(* CODESYS project plc_eposcmd.library
   Company: Maxon Motor
   Title: Maxon
   Version: 1.0.0.0

Project tree, tasks and I/O mapping:
  libraries: Tc2_System, * (Beckhoff Automation GmbH); Tc2_Standard, * (Beckhoff Automation GmbH)
  Data types/
  Global Variables/
    global variables Globale_Variablen
  POUs/
    Configuration/
      function block FB_GetCurrentRegulatorGain [ST]
      function block FB_GetEncoderParameter [ST]
      function block FB_GetMotorParameter [ST]
      function block FB_GetPositionRegulatorGain [ST]
      function block FB_GetVelocityRegulatorGain [ST]
      function block FB_SetCurrentRegulatorGain [ST]
      function block FB_SetEncoderParameter [ST]
      function block FB_SetMotorParameter [ST]
      function block FB_SetPositionRegulatorGain [ST]
      function block FB_SetVelocityRegulatorGain [ST]
    CurrentMode/
      function block FB_GetCurrentMust [ST]
      function block FB_SetCurrentMust [ST]
    HomingMode/
      function block FB_FindHome [ST]
      function block FB_GetHomingParameter [ST]
      function block FB_SetHomingParameter [ST]
      function block FB_StopHoming [ST]
    InputsOutputs/
      function block FB_GetAllDigitalInputs [ST]
      function block FB_GetAllDigitalOutputs [ST]
      function block FB_GetAnalogInput [ST]
      function block FB_SetAllDigitalOutputs [ST]
    MotionInfo/
      function block FB_GetCurrentIs [ST]
      function block FB_GetMovementState [ST]
      function block FB_GetPositionIs [ST]
      function block FB_GetVelocityIs [ST]
    PositionMode/
      function block FB_GetPositionMust [ST]
      function block FB_SetPositionMust [ST]
    ProfilePositionMode/
      function block FB_GetPositionProfile [ST]
      function block FB_GetTargetPosition [ST]
      function block FB_HaltPositionMovement [ST]
      function block FB_MoveToPosition [ST]
      function block FB_SetPositionProfile [ST]
    ProfileVelocityMode/
      function block FB_GetTargetVelocity [ST]
      function block FB_GetVelocityProfile [ST]
      function block FB_HaltVelocityMovement [ST]
      function block FB_MoveWithVelocity [ST]
      function block FB_SetVelocityProfile [ST]
    StateMachine/
      function block FB_ClearFault [ST]
      function block FB_GetDisableState [ST]
      function block FB_GetEnableState [ST]
      function block FB_GetFaultState [ST]
      function block FB_GetOperationMode [ST]
      function block FB_GetQuickStopState [ST]
      function block FB_SetDisableState [ST]
      function block FB_SetEnableState [ST]
      function block FB_SetOperationMode [ST]
      function block FB_SetQuickStopState [ST]
    Utilities/
      function block FB_GetObject [ST]
      function block FB_GetVersion [ST]
      function block FB_Restore [ST]
      function block FB_SetObject [ST]
      function block FB_Store [ST]
    VelocityMode/
      function block FB_GetVelocityMust [ST]
      function block FB_SetVelocityMust [ST]
  Visualizations/
*)

// Global Variables/Globale_Variablen
{attribute 'Tc2GvlVarNames'}
VAR_GLOBAL

END_VAR

// POUs/StateMachine/FB_ClearFault
FUNCTION_BLOCK FB_ClearFault
(*************************************************************************************************************************************
**	maxon motor ag
**	elektronik & systemtechnik
**	all rights reserved
**************************************************************************************************************************************
**	Summary :		Clear Error
**
**	Remarks : 	
**
**	Created under :	TwinCAT V 2.9.0 (Build 514)
**************************************************************************************************************************************
**	History : 
**	13.10.2003 	| 	san		Beta Version 0.10
**
*************************************************************************************************************************************)
VAR_INPUT
	ADSNetId		: STRING; 	(* Adresses the FC5101 or other Beckhoff CANOpen Masters.
								Can be empty if only local single channel card is present  *)
	NodeId			: INT;		(* Represents the node adress witch is found on Dip Switch of Device *)
	Write			: BOOL;		(* a rising edge starts writing *)

END_VAR
VAR_OUTPUT

	Done			: BOOL;		(* Done Flag is set when Function has done *)
	Err				: BOOL;		(* Err Flag is TRUE if an Error has accured, see Errno for more Details *)
	ErrNo			: UDINT;		(* Contains detailed Error Information *)
END_VAR
VAR
	iStep			: INT;
	WriteObj			: ADSWRITE;
	Controlword		: UINT	:= 16#0080;
	Multiplexor		: UDINT;		(* Gives Index and Subindex of actual Object *)
END_VAR

CASE iStep OF

1:	(* Init *)
	Write := FALSE;
	Done := FALSE;
	Err := FALSE;
	ErrNo := 0;
	WriteObj(WRITE := FALSE);
	iStep := 100;

100:	(* Write Controlword *)
	WriteObj(
		NETID := ADSNetId,
		PORT := 16#1000 + NodeId,
		IDXGRP := 16#6040,
		IDXOFFS := 0,
		LEN := 2,
		SRCADDR := ADR(Controlword),
		WRITE := TRUE,
		TMOUT := t#100ms);
	iStep := 101;
101:  WriteObj();
	IF NOT WriteObj.Busy THEN
		iStep := 102 ;
	END_IF
102:	IF WriteObj.Err THEN
		iStep := 0;
		ErrNo := WriteObj.ErrId;
		Multiplexor := 16#604000;
		Err := TRUE;
	ELSE
		iStep := 0;
	END_IF;
	Done := TRUE;

ELSE
	IF Write THEN
		iStep := 1;
		Done := FALSE;
	END_IF;
END_CASE;

END_FUNCTION_BLOCK

// POUs/HomingMode/FB_FindHome
FUNCTION_BLOCK FB_FindHome
(*************************************************************************************************************************************
**	maxon motor ag
**	elektronik & systemtechnik
**	all rights reserved
**************************************************************************************************************************************
**	Summary :		Find Home
**
**	Remarks : 	
**
**	Created under :	TwinCAT V 2.9.0 (Build 514)
**************************************************************************************************************************************
**	History : 
**	16.09.2003 	| 	san		Beta Version 0.10
**	21.11.2003	|	san		Beta Version 0.20 remove wait for status
**	03.02.2004	|	san		Bugfix set Done flag at the end
**
*************************************************************************************************************************************)
VAR_INPUT
	ADSNetId			: STRING; 	(* Adresses the FC5101 or other Beckhoff CANOpen Masters.
								Can be empty if only local single channel card is present  *)
	NodeId				: INT;		(* Represents the node adress witch is found on Dip Switch of Device *)
	Write				: BOOL;		(* a rising edge starts writing *)

	HomingMethod		: SINT;		(*see VAR CONSTANT *)
END_VAR
VAR_OUTPUT

	Done				: BOOL;		(* Done Flag is set when Function has done *)
	Err					: BOOL;		(* Err Flag is TRUE if an Error has accured, see Errno for more Details *)
	ErrNo				: UDINT;		(* Contains detailed Error Information *)
END_VAR
VAR
	iStep				: INT;
	WriteHomingMethod	: ADSWRITE;
	WriteCw				: ADSWRITE;
	ReadStatus			: ADSREAD;
	Controlword			: UINT;
	Statusword			: UINT;
	Multiplexor			: UDINT;		(* Gives Index and Subindex of actual Object *)
END_VAR

(*
VAR CONSTANT 
	cNegativeLimitSwitch						: SINT := 17;
	cPositiveLimitSwitch						: SINT := 18;
	cHomeSwitchPositiveSpeed				: SINT := 23;
	cHomeSwitchNegativeSpeed				: SINT := 27;
	cCurrentThresholdPositiveSpeed			: SINT := -3;
	cCurrentThresholdNegativeSpeed			: SINT := -4;
	cIndexPositiveSpeed						: SINT := 34;
	cIndexNegativeSpeed						: SINT := 33;
	cNegativeLimitSwitchAndIndex				: SINT := 1;
	cPositiveLimitSwitchAndIndex				: SINT := 2;
	cHomeSwitchPositiveSpeedAndIndex		: SINT := 7;
	cHomeSwitchNegativeSpeedAndIndex		: SINT := 11;
	cCurrentThresholdPositiveSpeedAndIndex	: SINT := -1;
	cCurrentThresholdNegativeSpeedAndIndex	: SINT := -2;
	cActualPositon							: SINT := 35;

END_VAR 
*)

CASE iStep OF

1:	(* Init *)
	Write := FALSE;
	Done := FALSE;
	Err := FALSE;
	ErrNo := 0;
	WriteHomingMethod(WRITE := FALSE);
	WriteCw(WRITE := FALSE);
	ReadStatus(READ := FALSE);
	iStep := 100;

100:	(* Write  Homing Method *)
	WriteHomingMethod(
		NETID := ADSNetId,
		PORT := 16#1000 + NodeId,
		IDXGRP := 16#6098,
		IDXOFFS := 0,
		LEN := 1,
		SRCADDR := ADR(HomingMethod),
		WRITE := TRUE,
		TMOUT := t#100ms);
	iStep := 101;
101:  WriteHomingMethod();
	IF NOT WriteHomingMethod.Busy THEN
		iStep := 102 ;
	END_IF
102:	IF WriteHomingMethod.Err THEN
		iStep := 0;
		ErrNo := WriteHomingMethod.ErrId;
		Multiplexor := 16#609800;
		Err := TRUE;
	ELSE
		iStep := 200;
	END_IF

200:	(* Write  Controlword Reset *)
	Controlword := 16#000F;
	WriteCw(
		NETID := ADSNetId,
		PORT := 16#1000 + NodeId,
		IDXGRP := 16#6040,
		IDXOFFS := 0,
		LEN := 2,
		SRCADDR := ADR(Controlword),
		WRITE := TRUE,
		TMOUT := t#100ms);
	iStep := 201;
201:  WriteCw();
	IF NOT WriteCw.Busy THEN
		iStep := 202 ;
	END_IF
202:	IF WriteCw.Err THEN
		iStep := 0;
		ErrNo := WriteCw.ErrId;
		Multiplexor := 16#604000;
		Err := TRUE;
	ELSE
		iStep := 300;
		WriteCw(WRITE := FALSE);
	END_IF

300:	(* Write  Controlword Start *)

	Controlword := 16#001F;
	WriteCw(
		NETID := ADSNetId,
		PORT := 16#1000 + NodeId,
		IDXGRP := 16#6040,
		IDXOFFS := 0,
		LEN := 2,
		SRCADDR := ADR(Controlword),
		WRITE := TRUE,
		TMOUT := t#100ms);
	iStep := 301;
301:  WriteCw();
	IF NOT WriteCw.Busy THEN
		iStep := 302 ;
	END_IF
302:	IF WriteCw.Err THEN
		iStep := 0;
		ErrNo := WriteCw.ErrId;
		Multiplexor := 16#604000;
		Err := TRUE;
	ELSE
		iStep := 0;
	END_IF
	Done := TRUE;
ELSE
	IF Write THEN
		iStep := 1;
		Done := FALSE;
	END_IF;
END_CASE;

END_FUNCTION_BLOCK

// POUs/InputsOutputs/FB_GetAllDigitalInputs
FUNCTION_BLOCK FB_GetAllDigitalInputs
(*************************************************************************************************************************************
**	maxon motor ag
**	elektronik & systemtechnik
**	all rights reserved
**************************************************************************************************************************************
**	Summary :		Read Digital Inputs
**
**	Remarks : 	
**
**	Created under :	TwinCAT V 2.9.0 (Build 514)
**************************************************************************************************************************************
**	History : 
**	16.09.2003 	| 	san		Beta Version 0.10
**	21.11.2003	|	san		Beta Version 0.20 firmware changes
**
*************************************************************************************************************************************)
VAR_INPUT
	ADSNetId		: STRING; 	(* Adresses the FC5101 or other Beckhoff CANOpen Masters.
								Can be empty if only local single channel card is present  *)
	NodeId			: INT;		(* Represents the node adress witch is found on Dip Switch of Device *)
	Read			: BOOL;		(* a rising edge start the reading *)
END_VAR
VAR_OUTPUT
	Done			: BOOL;		(* DataValid Flag is TRUE if Data were available *)
	Err				: BOOL;		(* Err Flag is TRUE if an Error has accured, see Errno for more Details *)
	ErrNo			: UDINT;		(* Contains detailed Error Information *)

	Inputs			: UINT;		(* Digital Inputs *)
END_VAR
VAR
	iStep			: INT;
	ReadObj			: ADSREAD;
	ODIdx			: UINT			:= 16#2071;
	Multiplexor		: UDINT;		(* Gives Index and Subindex of actual Object *)
END_VAR

CASE iStep OF

1:	(* Init *)
	Read := FALSE;
	Done := FALSE;
	Err := FALSE;
	ErrNo := 0;
	ReadObj(READ := FALSE);
	iStep := 100;

100:	(* Read Object *)
	ReadObj(
		NETID := ADSNetId,
		PORT := 16#1000 + NodeId,
		IDXGRP := ODIdx,
		IDXOFFS := 1,
		LEN := 2,
		DESTADDR := ADR(Inputs),
		READ := TRUE,
		TMOUT := t#100ms);
	iStep := 101;
101:  ReadObj();
	IF NOT ReadObj.Busy THEN
		iStep := 102 ;
	END_IF
102:	IF ReadObj.Err THEN
		iStep := 0;
		ErrNo := ReadObj.ErrId;
		Multiplexor := ODIdx * 256; (* Shift of 8 *)
		Err := TRUE;
	ELSE
		iStep := 0;
	END_IF;
	Done := TRUE;

ELSE
	IF Read THEN
		iStep := 1;
		Done := FALSE;
	END_IF;
END_CASE;

END_FUNCTION_BLOCK

// POUs/InputsOutputs/FB_GetAllDigitalOutputs
FUNCTION_BLOCK FB_GetAllDigitalOutputs
(*************************************************************************************************************************************
**	maxon motor ag
**	elektronik & systemtechnik
**	all rights reserved
**************************************************************************************************************************************
**	Summary :		Get all Digital Outputs
**
**	Remarks : 	
**
**	Created under :	TwinCAT V 2.9.0 (Build 514)
**************************************************************************************************************************************
**	History : 
**	16.09.2003 	| 	san		Beta Version 0.10
**	21.11.2003	|	san		Beta Version 0.20 firmware changes
**
*************************************************************************************************************************************)
VAR_INPUT
	ADSNetId		: STRING; 	(* Adresses the FC5101 or other Beckhoff CANOpen Masters.
								Can be empty if only local single channel card is present  *)
	NodeId			: INT;		(* Represents the node adress witch is found on Dip Switch of Device *)
	Write			: BOOL;		(* a rising edge starts writing *)

END_VAR
VAR_OUTPUT
	Done			: BOOL;		(* Done Flag is set when Function has done *)
	Err				: BOOL;		(* Err Flag is TRUE if an Error has accured, see Errno for more Details *)
	ErrNo			: UDINT;		(* Contains detailed Error Information *)

	Outputs			: UINT;
END_VAR
VAR
	iStep			: INT;
	ReadObj			: ADSREAD;
	ODIdx			: UINT			:= 16#2078;
	ODSubidx		: UINT			:= 1;
	Multiplexor		: UDINT;		(* Gives Index and Subindex of actual Object *)
END_VAR

CASE iStep OF

1:	(* Init *)
	Write := FALSE;
	Done := FALSE;
	Err := FALSE;
	ErrNo := 0;
	ReadObj(Read := FALSE);
	iStep := 100;

100:	(* Write Object *)
	ReadObj(
		NETID := ADSNetId,
		PORT := 16#1000 + NodeId,
		IDXGRP := ODIdx,
		IDXOFFS := ODSubidx,
		LEN := 2,
		DESTADDR := ADR(Outputs),
		READ := TRUE,
		TMOUT := t#100ms);
	iStep := 101;
101:  ReadObj();
	IF NOT ReadObj.Busy THEN
		iStep := 102 ;
	END_IF
102:	IF ReadObj.Err THEN
		iStep := 0;
		ErrNo := ReadObj.ErrId;
		Multiplexor := ODIdx * 256; (* Shift of 8 *)
		Multiplexor := Multiplexor + ODSubidx;
		Err := TRUE;
	ELSE
		iStep := 0;
	END_IF;
	Done := TRUE;

ELSE
	IF Write THEN
		iStep := 1;
		Done := FALSE;
	END_IF;
END_CASE;

END_FUNCTION_BLOCK

// POUs/InputsOutputs/FB_GetAnalogInput
FUNCTION_BLOCK FB_GetAnalogInput
(*************************************************************************************************************************************
**	maxon motor ag
**	elektronik & systemtechnik
**	all rights reserved
**************************************************************************************************************************************
**	Summary :		Read Analog Input Value
**
**	Remarks : 	
**
**	Created under :	TwinCAT V 2.9.0 (Build 514)
**************************************************************************************************************************************
**	History : 
**	16.09.2003 	| 	san		Beta Version 0.10
**	21.11.2003	|	san		Beta Version 0.20 firmware changes
**
*************************************************************************************************************************************)
VAR_INPUT
	ADSNetId		: STRING; 	(* Adresses the FC5101 or other Beckhoff CANOpen Masters.
								Can be empty if only local single channel card is present  *)
	NodeId			: INT;		(* Represents the node adress witch is found on Dip Switch of Device *)
	Read			: BOOL;		(* a rising edge start the reading *)

	Number			: UINT;		(* Analog Input Number *)
END_VAR
VAR_OUTPUT
	Done			: BOOL;		(* DataValid Flag is TRUE if Data were available *)
	Err				: BOOL;		(* Err Flag is TRUE if an Error has accured, see Errno for more Details *)
	ErrNo			: UDINT;		(* Contains detailed Error Information *)

	AnalogInput		: UINT;		(* Analog Input Value [mV] *)
END_VAR
VAR
	iStep			: INT;
	ReadObj			: ADSREAD;
	ODIdx			: UINT 	:= 16#207C;
	Multiplexor		: UDINT;		(* Gives Index and Subindex of actual Object *)
	ODSIdx			: UINT;
END_VAR

CASE iStep OF

1:	(* Init *)
	Read := FALSE;
	Done := FALSE;
	Err := FALSE;
	ErrNo := 0;
	ReadObj(READ := FALSE);
	IF (Number = 1) THEN
		ODSIdx := 1;
	ELSIF (Number = 2) THEN
		ODSIdx := 2;
	END_IF;
	iStep := 100;

100:	(* Read Object *)
	ReadObj(
		NETID := ADSNetId,
		PORT := 16#1000 + NodeId,
		IDXGRP := ODIdx,
		IDXOFFS := ODSIdx,
		LEN := 2,
		DESTADDR := ADR(AnalogInput),
		READ := TRUE,
		TMOUT := t#100ms);
	iStep := 101;
101:  ReadObj();
	IF NOT ReadObj.Busy THEN
		iStep := 102 ;
	END_IF
102:	IF ReadObj.Err THEN
		iStep := 0;
		ErrNo := ReadObj.ErrId;
		Multiplexor := ODIdx * 256; (* Shift of 8 *)
		Err := TRUE;
	ELSE
		iStep := 0;
	END_IF;
	Done := TRUE;

ELSE
	IF Read THEN
		iStep := 1;
		Done := FALSE;
	END_IF;
END_CASE;

END_FUNCTION_BLOCK

// POUs/MotionInfo/FB_GetCurrentIs
FUNCTION_BLOCK FB_GetCurrentIs
(*************************************************************************************************************************************
**	maxon motor ag
**	elektronik & systemtechnik
**	all rights reserved
**************************************************************************************************************************************
**	Summary :		Read Actual Value of Current
**
**	Remarks : 		
**
**	Created under :	TwinCAT V 2.9.0 (Build 514)
**************************************************************************************************************************************
**	History : 
**	13.10.2003 	| 	san		Beta Version 0.10
**
*************************************************************************************************************************************)
VAR_INPUT
	ADSNetId		: STRING; 	(* Adresses the FC5101 or other Beckhoff CANOpen Masters.
								Can be empty if only local single channel card is present  *)
	NodeId			: INT;		(* Represents the node adress witch is found on Dip Switch of Device *)
	Read			: BOOL;		(* a rising edge start the reading *)

END_VAR
VAR_OUTPUT
	Done			: BOOL;		(* DataValid Flag is TRUE if Data were available *)
	Err				: BOOL;		(* Err Flag is TRUE if an Error has accured, see Errno for more Details *)
	ErrNo			: UDINT;		(* Contains detailed Error Information *)

	CurrentIs			: INT;		(* Actual Value *)
END_VAR
VAR
	iStep			: INT;
	ReadObj			: ADSREAD;
	Multiplexor		: UDINT;		(* Gives Index and Subindex of actual Object *)
END_VAR

CASE iStep OF

1:	(* Init *)
	Read := FALSE;
	Done := FALSE;
	Err := FALSE;
	ErrNo := 0;
	ReadObj(READ := FALSE);
	iStep := 100;

100:	(* Read Object *)
	ReadObj(
		NETID := ADSNetId,
		PORT := 16#1000 + NodeId,
		IDXGRP := 16#6078,
		IDXOFFS := 0,
		LEN := 2,
		DESTADDR := ADR(CurrentIs),
		READ := TRUE,
		TMOUT := t#100ms);
	iStep := 101;
101:  ReadObj();
	IF NOT ReadObj.Busy THEN
		iStep := 102 ;
	END_IF
102:	IF ReadObj.Err THEN
		iStep := 0;
		ErrNo := ReadObj.ErrId;
		Multiplexor := 16#607800;
		Err := TRUE;
	ELSE
		iStep := 0;
	END_IF;
	Done := TRUE;

ELSE
	IF Read THEN
		iStep := 1;
		Done := FALSE;
	END_IF;
END_CASE;

END_FUNCTION_BLOCK

// POUs/CurrentMode/FB_GetCurrentMust
FUNCTION_BLOCK FB_GetCurrentMust
(*************************************************************************************************************************************
**	maxon motor ag
**	elektronik & systemtechnik
**	all rights reserved
**************************************************************************************************************************************
**	Summary :		Read Demand Value of Current
**
**	Remarks : 		
**
**	Created under :	TwinCAT V 2.9.0 (Build 514)
**************************************************************************************************************************************
**	History : 
**	13.10.2003 	| 	san		Beta Version 0.10
**
*************************************************************************************************************************************)
VAR_INPUT
	ADSNetId		: STRING; 	(* Adresses the FC5101 or other Beckhoff CANOpen Masters.
								Can be empty if only local single channel card is present  *)
	NodeId			: INT;		(* Represents the node adress witch is found on Dip Switch of Device *)
	Read			: BOOL;		(* a rising edge start the reading *)
END_VAR
VAR_OUTPUT
	Done			: BOOL;		(* DataValid Flag is TRUE if Data were available *)
	Err				: BOOL;		(* Err Flag is TRUE if an Error has accured, see Errno for more Details *)
	ErrNo			: UDINT;		(* Contains detailed Error Information *)

	CurrentMust		: INT;		(* Demand Value *)
END_VAR
VAR
	iStep			: INT;
	ReadObj			: ADSREAD;
	Multiplexor		: UDINT;		(* Gives Index and Subindex of actual Object *)
END_VAR

CASE iStep OF

1:	(* Init *)
	Read := FALSE;
	Done := FALSE;
	Err := FALSE;
	ErrNo := 0;
	ReadObj(READ := FALSE);
	iStep := 100;

100:	(* Read Object *)
	ReadObj(
		NETID := ADSNetId,
		PORT := 16#1000 + NodeId,
		IDXGRP := 16#2030,
		IDXOFFS := 0,
		LEN := 2,
		DESTADDR := ADR(CurrentMust),
		READ := TRUE,
		TMOUT := t#100ms);
	iStep := 101;
101:  ReadObj();
	IF NOT ReadObj.Busy THEN
		iStep := 102 ;
	END_IF
102:	IF ReadObj.Err THEN
		iStep := 0;
		ErrNo := ReadObj.ErrId;
		Multiplexor := 16#203000;
		Err := TRUE;
	ELSE
		iStep := 0;
	END_IF;
	Done := TRUE;

ELSE
	IF Read THEN
		iStep := 1;
		Done := FALSE;
	END_IF;
END_CASE;

END_FUNCTION_BLOCK

// POUs/Configuration/FB_GetCurrentRegulatorGain
FUNCTION_BLOCK FB_GetCurrentRegulatorGain
(*************************************************************************************************************************************
**	maxon motor ag
**	elektronik & systemtechnik
**	all rights reserved
**************************************************************************************************************************************
**	Summary :		Read Current Regulator Gains (PI)
**
**	Remarks : 		
**
**	Created under :	TwinCAT V 2.9.0 (Build 514)
**************************************************************************************************************************************
**	History : 
**	13.10.2003 	| 	san		Beta Version 0.10
**
*************************************************************************************************************************************)
VAR_INPUT
	ADSNetId		: STRING; 	(* Adresses the FC5101 or other Beckhoff CANOpen Masters.
								Can be empty if only local single channel card is present  *)
	NodeId			: INT;		(* Represents the node adress witch is found on Dip Switch of Device *)

	Read			: BOOL;		(* a rising edge starts reading *)
END_VAR
VAR_OUTPUT
	Done			: BOOL;		(* Done Flag is set when Function has done *)
	Err				: BOOL;		(* Err Flag is TRUE if an Error has accured, see Errno for more Details *)
	ErrNo			: UDINT;		(* Contains detailed Error Information *)

	P				: UINT;		(* Regulator P - Gain *)
	I				: UINT;		(* Regulator I - Gain  *)
END_VAR
VAR
	iStep			: INT;
	ReadP			: ADSREAD;
	ReadI			: ADSREAD;
	Multiplexor		: UDINT;		(* Gives Index and Subindex of actual Object *)
END_VAR

CASE iStep OF

1:	(* Init *)
	Read := FALSE;
	Done := FALSE;
	Err := FALSE;
	ErrNo := 0;
	ReadP(READ := FALSE);
	ReadI(READ := FALSE);
	iStep := 100;

100:	(* Read P - Gain *)
	ReadP(
		NETID := ADSNetId,
		PORT := 16#1000 + NodeId,
		IDXGRP := 16#60F6,
		IDXOFFS := 1,
		LEN := 2,
		DESTADDR := ADR(P),
		READ := TRUE,
		TMOUT := t#100ms);
	iStep := 101;
101:  ReadP();
	IF NOT ReadP.Busy THEN
		iStep := 102 ;
	END_IF
102:	IF ReadP.Err THEN
		iStep := 0;
		ErrNo := ReadP.ErrId;
		Multiplexor := 16#60F601;
		Err := TRUE;
	ELSE
		iStep := 200;
	END_IF

200:	(* Read I - Gain *)
	ReadI(
		NETID := ADSNetId,
		PORT := 16#1000 + NodeId,
		IDXGRP := 16#60F6,
		IDXOFFS := 2,
		LEN := 2,
		DESTADDR := ADR(I),
		READ := TRUE,
		TMOUT := t#100ms);
	iStep := 201;
201:  ReadI();
	IF NOT ReadI.Busy THEN
		iStep := 202 ;
	END_IF
202:	IF ReadI.Err THEN
		iStep := 0;
		ErrNo := ReadI.ErrId;
		Multiplexor := 16#60F602;
		Err := TRUE;
	ELSE
		iStep := 0;
	END_IF;
	Done := TRUE;

ELSE
	IF Read THEN
		iStep := 1;
		Done:= FALSE;
	END_IF;
END_CASE;

END_FUNCTION_BLOCK

// POUs/StateMachine/FB_GetDisableState
FUNCTION_BLOCK FB_GetDisableState
(*************************************************************************************************************************************
**	maxon motor ag
**	elektronik & systemtechnik
**	all rights reserved
**************************************************************************************************************************************
**	Summary :		Read Device Status
**
**	Remarks : 	
**
**	Created under :	TwinCAT V 2.9.0 (Build 514)
**************************************************************************************************************************************
**	History : 
**	30.09.2003 	| 	san		Beta Version 0.10
**
*************************************************************************************************************************************)
VAR_INPUT
	ADSNetId		: STRING; 	(* Adresses the FC5101 or other Beckhoff CANOpen Masters.
								Can be empty if only local single channel card is present  *)
	NodeId			: INT;		(* Represents the node adress witch is found on Dip Switch of Device *)
	Read			: BOOL;		(* a rising edge start the reading *)

END_VAR
VAR_OUTPUT
	Done			: BOOL;		(* DataValid Flag is TRUE if Data were available *)
	Err				: BOOL;		(* Err Flag is TRUE if an Error has accured, see Errno for more Details *)
	ErrNo			: UDINT;		(* Contains detailed Error Information *)

	IsDisabled		:BOOL;		(* TRUE:		Device is in Disable State
								    FALSE: 	Device is not in Disable State *)
END_VAR
VAR
	iStep			: INT;
	ReadObj			: ADSREAD;
	Multiplexor		: UDINT;		(* Gives Index and Subindex of actual Object *)
	Statusword		: UINT;		(* Device State *)

END_VAR

VAR CONSTANT
	cNotReadyToSwitchOn	:UINT := 16#0000;
	cSwitchOnDisabled		:UINT := 16#0040;
	cReadyToSwitchOn		:UINT := 16#0021;
	cSwitchedOn				:UINT := 16#0023;
	cOperationEnable			:UINT := 16#0027;
	cQuickStopActiv			:UINT := 16#0007;
	cFaultReactionActiv		:UINT := 16#000F;
	cFault					:UINT := 16#0008;

END_VAR

CASE iStep OF

1:	(* Init *)
	Read := FALSE;
	Done := FALSE;
	Err := FALSE;
	ErrNo := 0;
	ReadObj(READ := FALSE);
	iStep := 100;

100:	(* Read Status *)
	ReadObj(
		NETID := ADSNetId,
		PORT := 16#1000 + NodeId,
		IDXGRP := 16#6041,
		IDXOFFS := 0,
		LEN := 2,
		DESTADDR := ADR(Statusword),
		READ := TRUE,
		TMOUT := t#100ms);
	iStep := 101;
101:  ReadObj();
	IF NOT ReadObj.Busy THEN
		iStep := 102 ;
	END_IF
102:	IF ReadObj.Err THEN
		iStep := 0;
		ErrNo := ReadObj.ErrId;
		Multiplexor := 16#604100;
		Err := TRUE;
	ELSE
		iStep := 200;
	END_IF;


200:	IF (cNotReadyToSwitchOn = (UINT_TO_WORD(Statusword) AND 16#007F))  THEN
		IsDisabled := TRUE;
	ELSIF (cSwitchOnDisabled = (UINT_TO_WORD(Statusword) AND 16#007F))  THEN
		IsDisabled := TRUE;
	ELSIF (cReadyToSwitchOn = (UINT_TO_WORD(Statusword) AND 16#007F))  THEN
		IsDisabled := TRUE;
	ELSIF (cSwitchedOn = (UINT_TO_WORD(Statusword) AND 16#007F))  THEN
		IsDisabled := TRUE;
	ELSE
		IsDisabled := FALSE;
	END_IF;
	iStep := 0;
	Done := TRUE;

ELSE
	IF Read THEN
		iStep := 1;
		Done:= FALSE;
	END_IF;
END_CASE;

END_FUNCTION_BLOCK

// POUs/StateMachine/FB_GetEnableState
FUNCTION_BLOCK FB_GetEnableState
(*************************************************************************************************************************************
**	maxon motor ag
**	elektronik & systemtechnik
**	all rights reserved
**************************************************************************************************************************************
**	Summary :		Read Device Status
**
**	Remarks : 	
**
**	Created under :	TwinCAT V 2.9.0 (Build 514)
**************************************************************************************************************************************
**	History : 
**	30.09.2003 	| 	san		Beta Version 0.10
**
*************************************************************************************************************************************)
VAR_INPUT
	ADSNetId		: STRING; 	(* Adresses the FC5101 or other Beckhoff CANOpen Masters.
								Can be empty if only local single channel card is present  *)
	NodeId			: INT;		(* Represents the node adress witch is found on Dip Switch of Device *)
	Read			: BOOL;		(* a rising edge start the reading *)

END_VAR
VAR_OUTPUT
	Done			: BOOL;		(* DataValid Flag is TRUE if Data were available *)
	Err				: BOOL;		(* Err Flag is TRUE if an Error has accured, see Errno for more Details *)
	ErrNo			: UDINT;		(* Contains detailed Error Information *)

	IsEnabled		:BOOL;		(* TRUE:		Device is in Enable State
								    FALSE: 	Device is not in Enable State *)
END_VAR
VAR
	iStep			: INT;
	ReadObj			: ADSREAD;
	Multiplexor		: UDINT;		(* Gives Index and Subindex of actual Object *)
	Statusword		: UINT;		(* Device State *)

END_VAR

VAR CONSTANT
	cNotReadyToSwitchOn	:UINT := 16#0000;
	cSwitchOnDisabled		:UINT := 16#0040;
	cReadyToSwitchOn		:UINT := 16#0021;
	cSwitchedOn				:UINT := 16#0023;
	cOperationEnable			:UINT := 16#0027;
	cQuickStopActiv			:UINT := 16#0007;
	cFaultReactionActiv		:UINT := 16#000F;
	cFault					:UINT := 16#0008;

END_VAR

CASE iStep OF

1:	(* Init *)
	Read := FALSE;
	Done := FALSE;
	Err := FALSE;
	ErrNo := 0;
	ReadObj(READ := FALSE);
	iStep := 100;

100:	(* Read Status *)
	ReadObj(
		NETID := ADSNetId,
		PORT := 16#1000 + NodeId,
		IDXGRP := 16#6041,
		IDXOFFS := 0,
		LEN := 2,
		DESTADDR := ADR(Statusword),
		READ := TRUE,
		TMOUT := t#100ms);
	iStep := 101;
101:  ReadObj();
	IF NOT ReadObj.Busy THEN
		iStep := 102 ;
	END_IF
102:	IF ReadObj.Err THEN
		iStep := 0;
		ErrNo := ReadObj.ErrId;
		Multiplexor := 16#604100;
		Err := TRUE;
	ELSE
		iStep := 200;
	END_IF;


200:	IF (cOperationEnable = (UINT_TO_WORD(Statusword) AND 16#006F))  THEN
		IsEnabled := TRUE;
	ELSE
		IsEnabled := FALSE;
	END_IF;
	iStep := 0;
	Done := TRUE;

ELSE
	IF Read THEN
		iStep := 1;
		Done:= FALSE;
	END_IF;
END_CASE;

END_FUNCTION_BLOCK

// POUs/Configuration/FB_GetEncoderParameter
FUNCTION_BLOCK FB_GetEncoderParameter
(*************************************************************************************************************************************
**	maxon motor ag
**	elektronik & systemtechnik
**	all rights reserved
**************************************************************************************************************************************
**	Summary :		Read Encoder Parameter
**
**	Remarks : 		
**
**	Created under:	TwinCAT V 2.9.0 (Build 514)
**************************************************************************************************************************************
**	History : 
**	13.10.2003 	| 	san		Beta Version 0.10
**	21.11.2003	|	san		Beta Version 0.20 changes new SensorType
**
*************************************************************************************************************************************)
VAR_INPUT
	ADSNetId		: STRING; 	(* Adresses the FC5101 or other Beckhoff CANOpen Masters.
								Can be empty if only local single channel card is present  *)
	NodeId			: INT;		(* Represents the node adress witch is found on Dip Switch of Device *)

	Read			: BOOL;		(* a rising edge starts reading *)
END_VAR
VAR_OUTPUT
	Done			: BOOL;		(* Done Flag is set when Function has done *)
	Err				: BOOL;		(* Err Flag is TRUE if an Error has accured, see Errno for more Details *)
	ErrNo			: UDINT;		(* Contains detailed Error Information *)

	Counts			: UINT;
	SensorType		: UINT;
END_VAR
VAR
	iStep			: INT;
	ReadInc			: ADSREAD;
	ReadSt			: ADSREAD;
	Multiplexor		: UDINT;		(* Gives Index and Subindex of actual Object *)
END_VAR

CASE iStep OF

1:	(* Init *)
	Read := FALSE;
	Done := FALSE;
	Err := FALSE;
	ErrNo := 0;
	ReadInc(READ := FALSE);
	ReadSt(READ := FALSE);
	iStep := 100;

100:	(* Read Increments *)
	ReadInc(
		NETID := ADSNetId,
		PORT := 16#1000 + NodeId,
		IDXGRP := 16#221001,
		IDXOFFS := 5,
		LEN := 2,
		DESTADDR := ADR(Counts),
		READ := TRUE,
		TMOUT := t#100ms);
	iStep := 101;
101:  ReadInc();
	IF NOT ReadInc.Busy THEN
		iStep := 102 ;
	END_IF
102:	IF ReadInc.Err THEN
		iStep := 0;
		ErrNo := ReadInc.ErrId;
		Multiplexor := 16#221001;
		Err := TRUE;
	ELSE
		iStep := 200;
	END_IF

200:	(* Read Sensor Type *)
	ReadInc(
		NETID := ADSNetId,
		PORT := 16#1000 + NodeId,
		IDXGRP := 16#2210,
		IDXOFFS := 2,
		LEN := 2,
		DESTADDR := ADR(SensorType),
		READ := TRUE,
		TMOUT := t#100ms);
	iStep := 201;
201:  ReadSt();
	IF NOT ReadSt.Busy THEN
		iStep := 202 ;
	END_IF
202:	IF ReadSt.Err THEN
		iStep := 0;
		ErrNo := ReadSt.ErrId;
		Multiplexor := 16#221002;
		Err := TRUE;
	ELSE
		iStep := 0;
	END_IF
	Done := TRUE;

ELSE
	IF Read THEN
		iStep := 1;
		Done := FALSE;
	END_IF;
END_CASE;

END_FUNCTION_BLOCK

// POUs/StateMachine/FB_GetFaultState
FUNCTION_BLOCK FB_GetFaultState
(*************************************************************************************************************************************
**	maxon motor ag
**	elektronik & systemtechnik
**	all rights reserved
**************************************************************************************************************************************
**	Summary :		Read Device Status
**
**	Remarks : 	
**
**	Created under :	TwinCAT V 2.9.0 (Build 514)
**************************************************************************************************************************************
**	History : 
**	30.09.2003 	| 	san		Beta Version 0.10
**
*************************************************************************************************************************************)
VAR_INPUT
	ADSNetId		: STRING; 	(* Adresses the FC5101 or other Beckhoff CANOpen Masters.
								Can be empty if only local single channel card is present  *)
	NodeId			: INT;		(* Represents the node adress witch is found on Dip Switch of Device *)
	Read			: BOOL;		(* a rising edge start the reading *)

END_VAR
VAR_OUTPUT
	Done			: BOOL;		(* DataValid Flag is TRUE if Data were available *)
	Err				: BOOL;		(* Err Flag is TRUE if an Error has accured, see Errno for more Details *)
	ErrNo			: UDINT;		(* Contains detailed Error Information *)

	IsInErrorState		:BOOL;		(* TRUE:		Device is in Error State
								    FALSE: 	Device is not in Error State *)
END_VAR
VAR
	iStep			: INT;
	ReadObj			: ADSREAD;
	Multiplexor		: UDINT;		(* Gives Index and Subindex of actual Object *)
	Statusword		: UINT;		(* Device State *)

END_VAR

VAR CONSTANT
	cNotReadyToSwitchOn	:UINT := 16#0000;
	cSwitchOnDisabled		:UINT := 16#0040;
	cReadyToSwitchOn		:UINT := 16#0021;
	cSwitchedOn				:UINT := 16#0023;
	cOperationEnable			:UINT := 16#0027;
	cQuickStopActiv			:UINT := 16#0007;
	cFaultReactionActiv		:UINT := 16#000F;
	cFault					:UINT := 16#0008;

END_VAR

CASE iStep OF

1:	(* Init *)
	Read := FALSE;
	Done := FALSE;
	Err := FALSE;
	ErrNo := 0;
	ReadObj(READ := FALSE);
	iStep := 100;

100:	(* Read Status *)
	ReadObj(
		NETID := ADSNetId,
		PORT := 16#1000 + NodeId,
		IDXGRP := 16#6041,
		IDXOFFS := 0,
		LEN := 2,
		DESTADDR := ADR(Statusword),
		READ := TRUE,
		TMOUT := t#100ms);
	iStep := 101;
101:  ReadObj();
	IF NOT ReadObj.Busy THEN
		iStep := 102 ;
	END_IF
102:	IF ReadObj.Err THEN
		iStep := 0;
		ErrNo := ReadObj.ErrId;
		Multiplexor := 16#604100;
		Err := TRUE;
	ELSE
		iStep := 200;
	END_IF;


200:	IF (cFault = (UINT_TO_WORD(Statusword) AND 16#007F)) OR (cFaultReactionActiv = (UINT_TO_WORD(Statusword) AND 16#007F))  THEN
		IsInErrorState := TRUE;
	ELSE
		IsInErrorState := FALSE;
	END_IF;
	iStep := 0;
	Done := TRUE;

ELSE
	IF Read THEN
		iStep := 1;
		Done:= FALSE;
	END_IF;
END_CASE;

END_FUNCTION_BLOCK

// POUs/HomingMode/FB_GetHomingParameter
FUNCTION_BLOCK FB_GetHomingParameter
(*************************************************************************************************************************************
**	maxon motor ag
**	elektronik & systemtechnik
**	all rights reserved
**************************************************************************************************************************************
**	Summary :		Get all Homing Parameter
**
**	Remarks : 	
**
**	Created under :	TwinCAT V 2.9.0 (Build 514)
**************************************************************************************************************************************
**	History : 
**	30.09.2003 	| 	san		Beta Version 0.10
**	04.02.2004	|	san		CurrentTreshold renamed with CurrentThreshold
**
*************************************************************************************************************************************)
VAR_INPUT
	ADSNetId			: STRING; 	(* Adresses the FC5101 or other Beckhoff CANOpen Masters.
								Can be empty if only local single channel card is present  *)
	NodeId				: INT;		(* Represents the node adress witch is found on Dip Switch of Device *)
	Read				: BOOL;		(* a rising edge starts writing *)

END_VAR
VAR_OUTPUT

	Done				: BOOL;		(* Done Flag is set when Function has done *)
	Err					: BOOL;		(* Err Flag is TRUE if an Error has accured, see Errno for more Details *)
	ErrNo				: UDINT;		(* Contains detailed Error Information *)

	HomingAcceleration	: UDINT;
	SpeedSwitch			: UDINT;
	SpeedIndex			: UDINT;
	HomeOffset			: DINT;
	CurrentThreshold		: UINT;
END_VAR
VAR
	iStep				: INT;
	ReadHomingMethod	: ADSREAD;
	ReadHomingAcc		: ADSREAD;
	ReadHomingSpeed	: ADSREAD;
	ReadSpeedIndex		: ADSREAD;
	ReadHomeOffset		: ADSREAD;
	ReadCurTreshold		: ADSREAD;
	Controlword			: UINT;
	Multiplexor			: UDINT;		(* Gives Index and Subindex of actual Object *)
END_VAR

VAR CONSTANT
	(* HomingMethod *)
	cNegativeLimitSwitch						: SINT := 17;
	cPositiveLimitSwitch						: SINT := 18;
	cHomeSwitchPositiveSpeed				: SINT := 23;
	cHomeSwitchNegativeSpeed				: SINT := 27;
	cCurrentThresholdPositiveSpeed			: SINT := -3;
	cCurrentThresholdNegativeSpeed			: SINT := -4;
	cIndexPositiveSpeed						: SINT := 34;
	cIndexNegativeSpeed						: SINT := 33;
	cNegativeLimitSwitchAndIndex				: SINT := 1;
	cPositiveLimitSwitchAndIndex				: SINT := 2;
	cHomeSwitchPositiveSpeedAndIndex		: SINT := 7;
	cHomeSwitchNegativeSpeedAndIndex		: SINT := 11;
	cCurrentThresholdPositiveSpeedAndIndex	: SINT := -1;
	cCurrentThresholdNegativeSpeedAndIndex	: SINT := -2;
	cActualPositon							: SINT := 35;

END_VAR

CASE iStep OF

1:	(* Init *)
	Read := FALSE;
	Done := FALSE;
	Err := FALSE;
	ErrNo := 0;
	ReadHomingMethod(READ := FALSE);
	ReadHomingAcc(READ := FALSE);
	ReadHomingSpeed(READ := FALSE);
	ReadHomeOffset(READ := FALSE);
	ReadCurTreshold(READ := FALSE);
	iStep := 100;

100:	(* Read  Speed Index *)
	ReadSpeedIndex(
		NETID := ADSNetId,
		PORT := 16#1000 + NodeId,
		IDXGRP := 16#6099,
		IDXOFFS := 2,
		LEN := 4,
		DESTADDR := ADR(SpeedIndex),
		READ := TRUE,
		TMOUT := t#100ms);
	iStep := 101;
101:  ReadSpeedIndex();
	IF NOT ReadSpeedIndex.Busy THEN
		iStep := 102 ;
	END_IF
102:	IF ReadSpeedIndex.Err THEN
		iStep := 0;
		ErrNo := ReadSpeedIndex.ErrId;
		Multiplexor := 16#609902;
		Err := TRUE;
	ELSE
		iStep := 200;
	END_IF

200:	(* Read  Homing Acceleration *)
	ReadHomingAcc(
		NETID := ADSNetId,
		PORT := 16#1000 + NodeId,
		IDXGRP := 16#609A,
		IDXOFFS := 0,
		LEN := 4,
		DESTADDR := ADR(HomingAcceleration),
		READ := TRUE,
		TMOUT := t#100ms);
	iStep := 201;
201:  ReadHomingAcc();
	IF NOT ReadHomingAcc.Busy THEN
		iStep := 202 ;
	END_IF
202:	IF ReadHomingAcc.Err THEN
		iStep := 0;
		ErrNo := ReadHomingAcc.ErrId;
		Multiplexor := 16#609A00;
		Err := TRUE;
	ELSE
		iStep := 300;
	END_IF

300:	(* Read Homing Speed *)
	ReadHomingSpeed(
		NETID := ADSNetId,
		PORT := 16#1000 + NodeId,
		IDXGRP := 16#6099,
		IDXOFFS := 1,
		LEN := 4,
		DESTADDR := ADR(SpeedSwitch),
		READ := TRUE,
		TMOUT := t#100ms);
	iStep := 301;
301:  ReadHomingSpeed();
	IF NOT ReadHomingSpeed.Busy THEN
		iStep := 302 ;
	END_IF
302:	IF ReadHomingSpeed.Err THEN
		iStep := 0;
		ErrNo := ReadHomingSpeed.ErrId;
		Multiplexor := 16#609900;
		Err := TRUE;
	ELSE
		iStep := 400;
	END_IF

400:	(* Read  Homing Offset *)
	ReadHomeOffset(
		NETID := ADSNetId,
		PORT := 16#1000 + NodeId,
		IDXGRP := 16#607C,
		IDXOFFS := 0,
		LEN := 4,
		DESTADDR := ADR(HomeOffset),
		READ := TRUE,
		TMOUT := t#100ms);
	iStep := 401;
401:  ReadHomeOffset();
	IF NOT ReadHomeOffset.Busy THEN
		iStep := 402 ;
	END_IF
402:	IF ReadHomeOffset.Err THEN
		iStep := 0;
		ErrNo := ReadHomeOffset.ErrId;
		Multiplexor := 16#607C00;
		Err := TRUE;
	ELSE
		iStep := 500;
	END_IF

500:	(* Read  Current Treshold *)
	ReadCurTreshold(
		NETID := ADSNetId,
		PORT := 16#1000 + NodeId,
		IDXGRP := 16#2080,
		IDXOFFS := 0,
		LEN := 2,
		DESTADDR := ADR(CurrentThreshold),
		READ := TRUE,
		TMOUT := t#100ms);
	iStep := 501;
501:  ReadCurTreshold();
	IF NOT ReadCurTreshold.Busy THEN
		iStep := 502 ;
	END_IF
502:	IF ReadCurTreshold.Err THEN
		iStep := 0;
		ErrNo := ReadCurTreshold.ErrId;
		Multiplexor := 16#208000;
		Err := TRUE;
	ELSE
		iStep := 0;
	END_IF
	Done := TRUE;

ELSE
	IF Read THEN
		iStep := 1;
		Done := FALSE;
	END_IF;
END_CASE;

END_FUNCTION_BLOCK

// POUs/Configuration/FB_GetMotorParameter
FUNCTION_BLOCK FB_GetMotorParameter
(*************************************************************************************************************************************
**	maxon motor ag
**	elektronik & systemtechnik
**	all rights reserved
**************************************************************************************************************************************
**	Summary :		Read Motor Parameter
**
**	Remarks : 		
**
**	Created under :	TwinCAT V 2.9.0 (Build 514)
**************************************************************************************************************************************
**	History : 
**	13.10.2003 	| 	san		Beta Version 0.10
**	21.11.2003	|	san		Beta Version 0.20 firmware changes in object 6410
**
*************************************************************************************************************************************)
VAR_INPUT
	ADSNetId		: STRING; 	(* Adresses the FC5101 or other Beckhoff CANOpen Masters.
								Can be empty if only local single channel card is present  *)
	NodeId			: INT;		(* Represents the node adress witch is found on Dip Switch of Device *)

	Read			: BOOL;		(* a rising edge starts writing *)
END_VAR
VAR_OUTPUT
	Done			: BOOL;		(* Done Flag is set when Function has done *)
	Err				: BOOL;		(* Err Flag is TRUE if an Error has accured, see Errno for more Details *)
	ErrNo			: UDINT;		(* Contains detailed Error Information *)

	MotorType			: INT;		(*    10: Ec Motor	(Brushless Motor)
										1: Dc Motor	(Brushed Motor) *)

	ContinuousCurrent				: UINT;		(* Continuous Current *)
	PeakCurrent					: UINT;		(* Peak Current (normaly 2 * Icont) *)
	PolePair						: USINT;		(* Motor Pole Pair  *)
	ThermalTimeConstant			: UINT;		(* Thermal Time Constant *)
END_VAR
VAR
	iStep			: INT;
	ReadMTyp		: ADSREAD;
	ReadIcont		: ADSREAD;
	ReadIpeak		: ADSREAD;
	ReadPolePair	: ADSREAD;
	ReadTt			: ADSREAD;
	Multiplexor		: UDINT;		(* Gives Index and Subindex of actual Object *)
END_VAR

CASE iStep OF

1:	(* Init *)
	Read := FALSE;
	Done := FALSE;
	Err := FALSE;
	ErrNo := 0;
	ReadMTyp(READ := FALSE);
	ReadIcont(READ := FALSE);
	ReadIpeak(READ := FALSE);
	ReadPolePair(READ := FALSE);
	ReadTt(READ := FALSE);
	iStep := 100;

100:	(* Read MotorType *)
	ReadMTyp(
		NETID := ADSNetId,
		PORT := 16#1000 + NodeId,
		IDXGRP := 16#6402,
		IDXOFFS := 0,
		LEN := 2,
		DESTADDR := ADR(MotorType),
		READ := TRUE,
		TMOUT := t#100ms);
	iStep := 101;
101:  ReadMTyp();
	IF NOT ReadMTyp.Busy THEN
		iStep := 102 ;
	END_IF
102:	IF ReadMTyp.Err THEN
		iStep := 0;
		ErrNo := ReadMTyp.ErrId;
		Multiplexor := 16#640200;
		Err := TRUE;
	ELSE
		iStep := 200;
	END_IF

200:	(* Read Continuous Current*)
	ReadIcont(
		NETID := ADSNetId,
		PORT := 16#1000 + NodeId,
		IDXGRP := 16#6410,
		IDXOFFS := 1,
		LEN := 2,
		DESTADDR := ADR(ContinuousCurrent),
		READ := TRUE,
		TMOUT := t#100ms);
	iStep := 201;
201:  ReadIcont();
	IF NOT ReadIcont.Busy THEN
		iStep := 202 ;
	END_IF
202:	IF ReadIcont.Err THEN
		iStep := 0;
		ErrNo := ReadIcont.ErrId;
		Multiplexor := 16#641001;
		Err := TRUE;
	ELSE
		iStep := 300;
	END_IF

300:	(* Read Peak Current *)
	ReadIpeak(
		NETID := ADSNetId,
		PORT := 16#1000 + NodeId,
		IDXGRP := 16#6410,
		IDXOFFS := 2,
		LEN := 2,
		DESTADDR := ADR(PeakCurrent),
		READ := TRUE,
		TMOUT := t#100ms);
	iStep := 301;
301:  ReadIpeak();
	IF NOT ReadIpeak.Busy THEN
		iStep := 302 ;
	END_IF
302:	IF ReadIpeak.Err THEN
		iStep := 0;
		ErrNo := ReadIpeak.ErrId;
		Multiplexor := 16#641002;
		Err := TRUE;
	ELSE
		iStep := 400;
	END_IF

400:	(* Read Pole Pair *)
	ReadPolePair(
		NETID := ADSNetId,
		PORT := 16#1000 + NodeId,
		IDXGRP := 16#6410,
		IDXOFFS := 3,
		LEN := 1,
		DESTADDR := ADR(PolePair),
		READ := TRUE,
		TMOUT := t#100ms);
	iStep := 401;
401:  ReadPolePair();
	IF NOT ReadPolePair.Busy THEN
		iStep := 402 ;
	END_IF
402:	IF ReadPolePair.Err THEN
		iStep := 0;
		ErrNo := ReadPolePair.ErrId;
		Multiplexor := 16#641003;
		Err := TRUE;
	ELSE
		iStep := 600;
	END_IF

600:	(* Read Thermal Time Constant *)
	ReadTt(
		NETID := ADSNetId,
		PORT := 16#1000 + NodeId,
		IDXGRP := 16#6410,
		IDXOFFS := 5,
		LEN := 2,
		DESTADDR := ADR(ThermalTimeConstant),
		READ := TRUE,
		TMOUT := t#100ms);
	iStep := 601;
601:  ReadTt();
	IF NOT ReadTt.Busy THEN
		iStep := 602 ;
	END_IF
602:	IF ReadTt.Err THEN
		iStep := 0;
		ErrNo := ReadTt.ErrId;
		Multiplexor := 16#641005;
		Err := TRUE;
	ELSE
		iStep := 0;
	END_IF;
	Done := TRUE;

ELSE
	IF Read THEN
		iStep := 1;
		Done := FALSE;
	END_IF;
END_CASE;

END_FUNCTION_BLOCK

// POUs/MotionInfo/FB_GetMovementState
FUNCTION_BLOCK FB_GetMovementState
(*************************************************************************************************************************************
**	maxon motor ag
**	elektronik & systemtechnik
**	all rights reserved
**************************************************************************************************************************************
**	Summary :		Find Home
**
**	Remarks : 	
**
**	Created under :	TwinCAT V 2.9.0 (Build 514)
**************************************************************************************************************************************
**	History : 
**	30.09.2003 	| 	san		Beta Version 0.10
**	19.01.2004	|	san		Remove Write with Read Input
**
*************************************************************************************************************************************)
VAR_INPUT
	ADSNetId			: STRING; 	(* Adresses the FC5101 or other Beckhoff CANOpen Masters.
								Can be empty if only local single channel card is present  *)
	NodeId				: INT;		(* Represents the node adress witch is found on Dip Switch of Device *)
	Read				: BOOL;		(* a rising edge starts reading *)

END_VAR
VAR_OUTPUT

	Done				: BOOL;		(* Done Flag is set when Function has done *)
	Err					: BOOL;		(* Err Flag is TRUE if an Error has accured, see Errno for more Details *)
	ErrNo				: UDINT;		(* Contains detailed Error Information *)

	TargetReached		: BOOL;
END_VAR
VAR
	iStep				: INT;
	ReadStatus			: ADSREAD;
	Statusword			: UINT;
	Multiplexor			: UDINT;		(* Gives Index and Subindex of actual Object *)
END_VAR

CASE iStep OF

1:	(* Init *)
	Read := FALSE;
	Done := FALSE;
	Err := FALSE;
	ErrNo := 0;
	ReadStatus(READ := FALSE);
	iStep := 100;

100:	(* Read Status *)
	ReadStatus(
		NETID := ADSNetId,
		PORT := 16#1000 + NodeId,
		IDXGRP := 16#6041,
		IDXOFFS := 0,
		LEN := 2,
		DESTADDR := ADR(Statusword),
		READ := TRUE,
		TMOUT := t#100ms);
	iStep := 101;
101:  ReadStatus();
	IF NOT ReadStatus.Busy THEN
		iStep := 102 ;
	END_IF
102:	IF ReadStatus.Err THEN
		iStep := 0;
		ErrNo := ReadStatus.ErrId;
		Multiplexor := 16#6041000;
		Err := TRUE;
	ELSE
		IF ((UINT_TO_WORD(Statusword) AND 16#0400) =16#0400) THEN
			TargetReached := TRUE;
		ELSE
			TargetReached := FALSE;
		END_IF
		iStep := 0;
	END_IF
	Done := TRUE;

ELSE
	IF Read THEN
		iStep := 1;
		Done := FALSE;
		TargetReached:= FALSE;
	END_IF;
END_CASE;

END_FUNCTION_BLOCK

// POUs/Utilities/FB_GetObject
FUNCTION_BLOCK FB_GetObject
(*************************************************************************************************************************************
**	maxon motor ag
**	elektronik & systemtechnik
**	all rights reserved
**************************************************************************************************************************************
**	Summary :		Reads one Object from Object Dictionary
**
**	Remarks : 	
**
**	Created under :	TwinCAT V 2.9.0 (Build 514)
**************************************************************************************************************************************
**	History : 
**	13.10.2003 	| 	san		Beta Version 0.10
**	04.02.2004	|	san		ODIdx renamed witth ObjectIndex, ODSubidx renamed with ObjectSubindex
**
*************************************************************************************************************************************)
VAR_INPUT
	ADSNetId		: STRING; 	(* Adresses the FC5101 or other Beckhoff CANOpen Masters.
								Can be empty if only local single channel card is present  *)
	NodeId			: INT;		(* Represents the node adress witch is found on Dip Switch of Device *)
	Read			: BOOL;		(* a rising edge start the reading *)

	ObjectIndex		: UINT;		(* Object Dictionary Index *)
	ObjectSubindex	: USINT;		(* Object Dictionary Sub Index *)
	Len				: USINT;		(* Length of Object, Number of Bytes *)
END_VAR
VAR_OUTPUT
	Done			: BOOL;		(* DataValid Flag is TRUE if Data were available *)
	Err				: BOOL;		(* Err Flag is TRUE if an Error has accured, see Errno for more Details *)
	ErrNo			: UDINT;		(* Contains detailed Error Information *)

	Data			: UDINT;		(* Data Field *)
END_VAR
VAR
	iStep			: INT;
	ReadObj			: ADSREAD;
	Multiplexor		: UDINT;		(* Gives Index and Subindex of actual Object *)
END_VAR

CASE iStep OF

1:	(* Init *)
	Read := FALSE;
	Done := FALSE;
	Err := FALSE;
	ErrNo := 0;
	ReadObj(READ := FALSE);
	iStep := 100;

100:	(* Read Object *)
	ReadObj(
		NETID := ADSNetId,
		PORT := 16#1000 + NodeId,
		IDXGRP := ObjectIndex,
		IDXOFFS := ObjectSubindex,
		LEN := LEN,
		DESTADDR := ADR(Data),
		READ := TRUE,
		TMOUT := t#100ms);
	iStep := 101;
101:  ReadObj();
	IF NOT ReadObj.Busy THEN
		iStep := 102 ;
	END_IF
102:	IF ReadObj.Err THEN
		iStep := 0;
		ErrNo := ReadObj.ErrId;
		Multiplexor := ObjectIndex * 256; (* Shift of 8 *)
		Multiplexor := Multiplexor + ObjectSubindex;
		Err := TRUE;
	ELSE
		iStep := 0;
	END_IF;
	Done := TRUE;

ELSE
	IF Read THEN
		iStep := 1;
		Done := FALSE;
	END_IF;
END_CASE;

END_FUNCTION_BLOCK

// POUs/StateMachine/FB_GetOperationMode
FUNCTION_BLOCK FB_GetOperationMode
(*************************************************************************************************************************************
**	maxon motor ag
**	elektronik & systemtechnik
**	all rights reserved
**************************************************************************************************************************************
**	Summary :		Read Operation Mode
**
**	Remarks : 	
**
**	Created under :	TwinCAT V 2.9.0 (Build 514)
**************************************************************************************************************************************
**	History : 
**	13.10.2003 	| 	san		Beta Version 0.10
**	04.02.2004	|	san		type of Mode changed from USINT to SINT
**
*************************************************************************************************************************************)
VAR_INPUT
	ADSNetId		: STRING; 	(* Adresses the FC5101 or other Beckhoff CANOpen Masters.
								Can be empty if only local single channel card is present  *)
	NodeId			: INT;		(* Represents the node adress witch is found on Dip Switch of Device *)
	Read			: BOOL;		(* a rising edge start the reading *)

END_VAR
VAR_OUTPUT
	Done			: BOOL;		(* DataValid Flag is TRUE if Data were available *)
	Err				: BOOL;		(* Err Flag is TRUE if an Error has accured, see Errno for more Details *)
	ErrNo			: UDINT;		(* Contains detailed Error Information *)

	Mode			: SINT;		(* Operation Mode:
									16#01	= 	ProfilePositonMode
									16#03	= 	ProfileVelocityMode
									16#06	= 	HomingMode
									16#FF	= 	PositonMode
									16#FE	= 	VelocityMode
									16#FD	= 	CurrentMode
									 *)
END_VAR
VAR
	iStep			: INT;
	ReadObj			: ADSREAD;
	Multiplexor		: UDINT;		(* Gives Index and Subindex of actual Object *)
END_VAR

CASE iStep OF

1:	(* Init *)
	Read := FALSE;
	Done := FALSE;
	Err := FALSE;
	ErrNo := 0;
	ReadObj(READ := FALSE);
	iStep := 100;

100:	(* Read Status *)
	ReadObj(
		NETID := ADSNetId,
		PORT := 16#1000 + NodeId,
		IDXGRP := 16#6061,
		IDXOFFS := 0,
		LEN := 1,
		DESTADDR := ADR(Mode),
		READ := TRUE,
		TMOUT := t#100ms);
	iStep := 101;
101:  ReadObj();
	IF NOT ReadObj.Busy THEN
		iStep := 102 ;
	END_IF
102:	IF ReadObj.Err THEN
		iStep := 0;
		ErrNo := ReadObj.ErrId;
		Multiplexor := 16#606100;
		Err := TRUE;
	ELSE
		iStep := 0;
	END_IF;
	Done := TRUE;

ELSE
	IF Read THEN
		iStep := 1;
		Done:= FALSE;
	END_IF;
END_CASE;

END_FUNCTION_BLOCK

// POUs/MotionInfo/FB_GetPositionIs
FUNCTION_BLOCK FB_GetPositionIs
(*************************************************************************************************************************************
**	maxon motor ag
**	elektronik & systemtechnik
**	all rights reserved
**************************************************************************************************************************************
**	Summary :		Read Actual Value of Position
**
**	Remarks : 	
**
**	Created under :	TwinCAT V 2.9.0 (Build 514)
**************************************************************************************************************************************
**	History : 
**	13.10.2003 	| 	san		Beta Version 0.10
**
*************************************************************************************************************************************)
VAR_INPUT
	ADSNetId		: STRING; 	(* Adresses the FC5101 or other Beckhoff CANOpen Masters.
								Can be empty if only local single channel card is present  *)
	NodeId			: INT;		(* Represents the node adress witch is found on Dip Switch of Device *)
	Read			: BOOL;		(* a rising edge start the reading *)

END_VAR
VAR_OUTPUT
	Done			: BOOL;		(* DataValid Flag is TRUE if Data were available *)
	Err				: BOOL;		(* Err Flag is TRUE if an Error has accured, see Errno for more Details *)
	ErrNo			: UDINT;		(* Contains detailed Error Information *)

	PositionIs		: DINT;		(* Actual Value *)
END_VAR
VAR
	iStep			: INT;
	ReadObj			: ADSREAD;
	Multiplexor		: UDINT;		(* Gives Index and Subindex of actual Object *)
END_VAR

CASE iStep OF

1:	(* Init *)
	Read := FALSE;
	Done := FALSE;
	Err := FALSE;
	ErrNo := 0;
	ReadObj(READ := FALSE);
	iStep := 100;

100:	(* Read Object *)
	ReadObj(
		NETID := ADSNetId,
		PORT := 16#1000 + NodeId,
		IDXGRP := 16#6064,
		IDXOFFS := 0,
		LEN := 4,
		DESTADDR := ADR(PositionIs),
		READ := TRUE,
		TMOUT := t#100ms);
	iStep := 101;
101:  ReadObj();
	IF NOT ReadObj.Busy THEN
		iStep := 102 ;
	END_IF
102:	IF ReadObj.Err THEN
		iStep := 0;
		ErrNo := ReadObj.ErrId;
		Multiplexor := 16#606400;
		Err := TRUE;
	ELSE
		iStep := 0;
	END_IF;
	Done := TRUE;

ELSE
	IF Read THEN
		iStep := 1;
		Done := FALSE;
	END_IF;
END_CASE;

END_FUNCTION_BLOCK

// POUs/PositionMode/FB_GetPositionMust
FUNCTION_BLOCK FB_GetPositionMust
(*************************************************************************************************************************************
**	maxon motor ag
**	elektronik & systemtechnik
**	all rights reserved
**************************************************************************************************************************************
**	Summary :		Read Demand Value of Position
**
**	Remarks : 	
**
**	Created under :	TwinCAT V 2.9.0 (Build 514)
**************************************************************************************************************************************
**	History : 
**	13.10.2003 	| 	san		Beta Version 0.10
**
*************************************************************************************************************************************)
VAR_INPUT
	ADSNetId		: STRING; 	(* Adresses the FC5101 or other Beckhoff CANOpen Masters.
								Can be empty if only local single channel card is present  *)
	NodeId			: INT;		(* Represents the node adress witch is found on Dip Switch of Device *)
	Read			: BOOL;		(* a rising edge start the reading *)

END_VAR
VAR_OUTPUT
	Done			: BOOL;		(* DataValid Flag is TRUE if Data were available *)
	Err				: BOOL;		(* Err Flag is TRUE if an Error has accured, see Errno for more Details *)
	ErrNo			: UDINT;		(* Contains detailed Error Information *)

	PositionMust		: DINT;		(* Demand Value *)

END_VAR
VAR
	iStep			: INT;
	ReadObj			: ADSREAD;
	Multiplexor		: UDINT;		(* Gives Index and Subindex of actual Object *)
END_VAR

CASE iStep OF

1:	(* Init *)
	Read := FALSE;
	Done := FALSE;
	Err := FALSE;
	ErrNo := 0;
	ReadObj(READ := FALSE);
	iStep := 100;

100:	(* Read Object *)
	ReadObj(
		NETID := ADSNetId,
		PORT := 16#1000 + NodeId,
		IDXGRP := 16#2062,
		IDXOFFS := 0,
		LEN := 4,
		DESTADDR := ADR(PositionMust),
		READ := TRUE,
		TMOUT := t#100ms);
	iStep := 101;
101:  ReadObj();
	IF NOT ReadObj.Busy THEN
		iStep := 102 ;
	END_IF
102:	IF ReadObj.Err THEN
		iStep := 0;
		ErrNo := ReadObj.ErrId;
		Multiplexor := 16#206200;
		Err := TRUE;
	ELSE
		iStep := 0;
	END_IF;
	Done := TRUE;

ELSE
	IF Read THEN
		iStep := 1;
		Done := FALSE;
	END_IF;
END_CASE;

END_FUNCTION_BLOCK

// POUs/ProfilePositionMode/FB_GetPositionProfile
FUNCTION_BLOCK FB_GetPositionProfile
(*************************************************************************************************************************************
**	maxon motor ag
**	elektronik & systemtechnik
**	all rights reserved
**************************************************************************************************************************************
**	Summary :		Get Position Profile
**
**	Remarks : 		
**
**	Created under:	TwinCAT V 2.9.0 (Build 514)
**************************************************************************************************************************************
**	History : 
**	13.10.2003 	| 	san		Beta Version 0.10
**
*************************************************************************************************************************************)
VAR_INPUT
	ADSNetId		: STRING; 	(* Adresses the FC5101 or other Beckhoff CANOpen Masters.
								Can be empty if only local single channel card is present  *)
	NodeId			: INT;		(* Represents the node adress witch is found on Dip Switch of Device *)

	Read			: BOOL;		(* a rising edge starts reading *)

END_VAR
VAR_OUTPUT
	Done			: BOOL;		(* Done Flag is set when Function has done *)
	Err				: BOOL;		(* Err Flag is TRUE if an Error has accured, see Errno for more Details *)
	ErrNo			: UDINT;		(* Contains detailed Error Information *)

	ProfileVelocity	: UDINT;		(* Profile Velocity *)
	ProfileAcceleration: UDINT;		(* Profile Acceleration *)
	ProfileDeceleration: UDINT;		(* Profile Deceleration *)
END_VAR
VAR
	iStep			: INT;
	ReadVel			: ADSREAD;
	ReadAcc		: ADSREAD;
	ReadDec		: ADSREAD;
	Multiplexor		: UDINT;		(* Gives Index and Subindex of actual Object *)
END_VAR

CASE iStep OF

1:	(* Init *)
	Read := FALSE;
	Done := FALSE;
	Err := FALSE;
	ErrNo := 0;
	ReadVel(READ := FALSE);
	ReadAcc(READ := FALSE);
	ReadDec(READ := FALSE);
	iStep := 100;

100:	(* Profile Velocity *)
	ReadVel(
		NETID := ADSNetId,
		PORT := 16#1000 + NodeId,
		IDXGRP := 16#6081,
		IDXOFFS := 0,
		LEN := 4,
		DESTADDR := ADR(ProfileVelocity),
		READ := TRUE,
		TMOUT := t#100ms);
	iStep := 101;
101:  ReadVel();
	IF NOT ReadVel.Busy THEN
		iStep := 102 ;
	END_IF
102:	IF READVel.Err THEN
		iStep := 0;
		ErrNo := READVel.ErrId;
		Multiplexor := 16#608100;
		Err := TRUE;
	ELSE
		iStep := 200;
	END_IF

200:	(* Profile Acceleration *)
	ReadAcc(
		NETID := ADSNetId,
		PORT := 16#1000 + NodeId,
		IDXGRP := 16#6083,
		IDXOFFS := 0,
		LEN := 4,
		DESTADDR := ADR(ProfileAcceleration),
		READ := TRUE,
		TMOUT := t#100ms);
	iStep := 201;
201:  ReadAcc();
	IF NOT ReadAcc.Busy THEN
		iStep := 202 ;
	END_IF
202:	IF ReadAcc.Err THEN
		iStep := 0;
		ErrNo := ReadAcc.ErrId;
		Multiplexor := 16#608300;
		Err := TRUE;
	ELSE
		iStep := 300;
	END_IF

300:	(* Profile Deceleration *)
	ReadDec(
		NETID := ADSNetId,
		PORT := 16#1000 + NodeId,
		IDXGRP := 16#6084,
		IDXOFFS := 0,
		LEN := 4,
		DESTADDR := ADR(ProfileDeceleration),
		READ := TRUE,
		TMOUT := t#100ms);
	iStep := 301;
301:  ReadDec();
	IF NOT ReadDec.Busy THEN
		iStep := 302 ;
	END_IF
302:	IF ReadDec.Err THEN
		iStep := 0;
		ErrNo := ReadDec.ErrId;
		Multiplexor := 16#608400;
		Err := TRUE;
	ELSE
		iStep := 0;
	END_IF;
	Done := TRUE;

ELSE
	IF Read THEN
		iStep := 1;
		Done := FALSE;
	END_IF;
END_CASE;

END_FUNCTION_BLOCK

// POUs/Configuration/FB_GetPositionRegulatorGain
FUNCTION_BLOCK FB_GetPositionRegulatorGain
(*************************************************************************************************************************************
**	maxon motor ag
**	elektronik & systemtechnik
**	all rights reserved
**************************************************************************************************************************************
**	Summary :		Read Position Regulator Gains (PID)
**
**	Remarks : 		
**
**	Created under :	TwinCAT V 2.9.0 (Build 514)
**************************************************************************************************************************************
**	History : 
**	13.10.2003 	| 	san		Beta Version 0.10
**
*************************************************************************************************************************************)
VAR_INPUT
	ADSNetId		: STRING; 	(* Adresses the FC5101 or other Beckhoff CANOpen Masters.
								Can be empty if only local single channel card is present  *)
	NodeId			: INT;		(* Represents the node adress witch is found on Dip Switch of Device *)
	Read			: BOOL;		(* a rising edge starts reading *)
END_VAR
VAR_OUTPUT
	Done			: BOOL;		(* Done Flag is set when Function has done *)
	Err				: BOOL;		(* Err Flag is TRUE if an Error has accured, see Errno for more Details *)
	ErrNo			: UDINT;		(* Contains detailed Error Information *)

	P				: UINT;		(* Regulator P - Gain *)
	I				: UINT;		(* Regulator I - Gain  *)
	D				: UINT;		(* Regulator D - Gain *)
END_VAR
VAR
	iStep			: INT;
	ReadP			: ADSREAD;
	ReadI			: ADSREAD;
	ReadD			: ADSREAD;
	Multiplexor		: UDINT;		(* Gives Index and Subindex of actual Object *)
END_VAR

CASE iStep OF

1:	(* Init *)
	Read := FALSE;
	Done := FALSE;
	Err := FALSE;
	ErrNo := 0;
	ReadP(READ := FALSE);
	ReadI(READ := FALSE);
	ReadD(READ := FALSE);
	iStep := 100;

100:	(* Read P - Gain *)
	ReadP(
		NETID := ADSNetId,
		PORT := 16#1000 + NodeId,
		IDXGRP := 16#60FB,
		IDXOFFS := 1,
		LEN := 2,
		DESTADDR := ADR(P),
		READ := TRUE,
		TMOUT := t#100ms);
	iStep := 101;
101:  ReadP();
	IF NOT ReadP.Busy THEN
		iStep := 102 ;
	END_IF
102:	IF ReadP.Err THEN
		iStep := 0;
		ErrNo := ReadP.ErrId;
		Multiplexor := 16#60FB01;
		Err := TRUE;
	ELSE
		iStep := 200;
	END_IF

200:	(* Read I - Gain *)
	ReadI(
		NETID := ADSNetId,
		PORT := 16#1000 + NodeId,
		IDXGRP := 16#60FB,
		IDXOFFS := 2,
		LEN := 2,
		DESTADDR := ADR(I),
		READ := TRUE,
		TMOUT := t#100ms);
	iStep := 201;
201:  ReadI();
	IF NOT ReadI.Busy THEN
		iStep := 202 ;
	END_IF
202:	IF ReadI.Err THEN
		iStep := 0;
		ErrNo := ReadI.ErrId;
		Multiplexor := 16#60FB02;
		Err := TRUE;
	ELSE
		iStep := 300;
	END_IF

300:	(* Read D - Gain *)
	ReadD(
		NETID := ADSNetId,
		PORT := 16#1000 + NodeId,
		IDXGRP := 16#60FB,
		IDXOFFS := 3,
		LEN := 2,
		DESTADDR := ADR(D),
		READ := TRUE,
		TMOUT := t#100ms);
	iStep := 301;
301:  ReadD();
	IF NOT ReadD.Busy THEN
		iStep := 302 ;
	END_IF
302:	IF ReadD.Err THEN
		iStep := 0;
		ErrNo := ReadD.ErrId;
		Multiplexor := 16#60FB03;
		Err := TRUE;
	ELSE
		iStep := 0;
	END_IF;
	Done := TRUE;

ELSE
	IF Read THEN
		iStep := 1;
		Done := FALSE;
	END_IF;
END_CASE;

END_FUNCTION_BLOCK

// POUs/StateMachine/FB_GetQuickStopState
FUNCTION_BLOCK FB_GetQuickStopState
(*************************************************************************************************************************************
**	maxon motor ag
**	elektronik & systemtechnik
**	all rights reserved
**************************************************************************************************************************************
**	Summary :		Read Device Status
**
**	Remarks : 	
**
**	Created under :	TwinCAT V 2.9.0 (Build 514)
**************************************************************************************************************************************
**	History : 
**	30.09.2003 	| 	san		Beta Version 0.10
**
*************************************************************************************************************************************)
VAR_INPUT
	ADSNetId		: STRING; 	(* Adresses the FC5101 or other Beckhoff CANOpen Masters.
								Can be empty if only local single channel card is present  *)
	NodeId			: INT;		(* Represents the node adress witch is found on Dip Switch of Device *)
	Read			: BOOL;		(* a rising edge start the reading *)

END_VAR
VAR_OUTPUT
	Done			: BOOL;		(* DataValid Flag is TRUE if Data were available *)
	Err				: BOOL;		(* Err Flag is TRUE if an Error has accured, see Errno for more Details *)
	ErrNo			: UDINT;		(* Contains detailed Error Information *)

	IsStoped			:BOOL;		(* TRUE:		Device is in Quick Stop State
								    FALSE: 	Device is not in Quick Stop State *)
END_VAR
VAR
	iStep			: INT;
	ReadObj			: ADSREAD;
	Multiplexor		: UDINT;		(* Gives Index and Subindex of actual Object *)
	Statusword		: UINT;		(* Device State *)
END_VAR

VAR CONSTANT
	cNotReadyToSwitchOn	:UINT := 16#0000;
	cSwitchOnDisabled		:UINT := 16#0040;
	cReadyToSwitchOn		:UINT := 16#0021;
	cSwitchedOn				:UINT := 16#0023;
	cOperationEnable			:UINT := 16#0027;
	cQuickStopActiv			:UINT := 16#0007;
	cFaultReactionActiv		:UINT := 16#000F;
	cFault					:UINT := 16#0008;

END_VAR

CASE iStep OF

1:	(* Init *)
	Read := FALSE;
	Done := FALSE;
	Err := FALSE;
	ErrNo := 0;
	ReadObj(READ := FALSE);
	iStep := 100;

100:	(* Read Status *)
	ReadObj(
		NETID := ADSNetId,
		PORT := 16#1000 + NodeId,
		IDXGRP := 16#6041,
		IDXOFFS := 0,
		LEN := 2,
		DESTADDR := ADR(Statusword),
		READ := TRUE,
		TMOUT := t#100ms);
	iStep := 101;
101:  ReadObj();
	IF NOT ReadObj.Busy THEN
		iStep := 102 ;
	END_IF
102:	IF ReadObj.Err THEN
		iStep := 0;
		ErrNo := ReadObj.ErrId;
		Multiplexor := 16#604100;
		Err := TRUE;
	ELSE
		iStep := 200;
	END_IF;


200:	IF cQuickStopActiv = (UINT_TO_WORD(Statusword) AND 16#006F) THEN
		IsStoped := TRUE;
	ELSE
		IsStoped := FALSE;
	END_IF;
	iStep := 0;
	Done := TRUE;

ELSE
	IF Read THEN
		iStep := 1;
		Done:= FALSE;
	END_IF;
END_CASE;

END_FUNCTION_BLOCK

// POUs/ProfilePositionMode/FB_GetTargetPosition
FUNCTION_BLOCK FB_GetTargetPosition
(*************************************************************************************************************************************
**	maxon motor ag
**	elektronik & systemtechnik
**	all rights reserved
**************************************************************************************************************************************
**	Summary :		Read Target Value of Position
**
**	Remarks : 	
**
**	Created under :	TwinCAT V 2.9.0 (Build 514)
**************************************************************************************************************************************
**	History : 
**	13.10.2003 	| 	san		Beta Version 0.10
**
*************************************************************************************************************************************)
VAR_INPUT
	ADSNetId		: STRING; 	(* Adresses the FC5101 or other Beckhoff CANOpen Masters.
								Can be empty if only local single channel card is present  *)
	NodeId			: INT;		(* Represents the node adress witch is found on Dip Switch of Device *)

	Read			: BOOL;		(* a rising edge start the reading *)

END_VAR
VAR_OUTPUT
	Done			: BOOL;		(* DataValid Flag is TRUE if Data were available *)
	Err				: BOOL;		(* Err Flag is TRUE if an Error has accured, see Errno for more Details *)
	ErrNo			: UDINT;		(* Contains detailed Error Information *)

	TargetPosition	: DINT;		(* Target Value *)

END_VAR
VAR
	iStep			: INT;
	ReadObj			: ADSREAD;
	Multiplexor		: UDINT;		(* Gives Index and Subindex of actual Object *)
END_VAR

CASE iStep OF

1:	(* Init *)
	Read := FALSE;
	Done:= FALSE;
	Err := FALSE;
	ErrNo := 0;
	ReadObj(READ := FALSE);
	iStep := 100;

100:	(* Read Object *)
	ReadObj(
		NETID := ADSNetId,
		PORT := 16#1000 + NodeId,
		IDXGRP := 16#607A,
		IDXOFFS := 0,
		LEN := 4,
		DESTADDR := ADR(TargetPosition),
		READ := TRUE,
		TMOUT := t#100ms);
	iStep := 101;
101:  ReadObj();
	IF NOT ReadObj.Busy THEN
		iStep := 102 ;
	END_IF
102:	IF ReadObj.Err THEN
		iStep := 0;
		ErrNo := ReadObj.ErrId;
		Multiplexor := 16#607A00;
		Err := TRUE;
	ELSE
		iStep := 0;
	END_IF;
	Done := TRUE;

ELSE
	IF Read THEN
		iStep := 1;
		Done := FALSE;
	END_IF;
END_CASE;

END_FUNCTION_BLOCK

// POUs/ProfileVelocityMode/FB_GetTargetVelocity
FUNCTION_BLOCK FB_GetTargetVelocity
(*************************************************************************************************************************************
**	maxon motor ag
**	elektronik & systemtechnik
**	all rights reserved
**************************************************************************************************************************************
**	Summary :		Read Target Value of Velocity
**
**	Remarks : 	
**
**	Created under :	TwinCAT V 2.9.0 (Build 514)
**************************************************************************************************************************************
**	History : 
**	13.10.2003 	| 	san		Beta Version 0.10
**
*************************************************************************************************************************************)
VAR_INPUT
	ADSNetId		: STRING; 	(* Adresses the FC5101 or other Beckhoff CANOpen Masters.
								Can be empty if only local single channel card is present  *)
	NodeId			: INT;		(* Represents the node adress witch is found on Dip Switch of Device *)
	Read			: BOOL;		(* a rising edge start the reading *)

END_VAR
VAR_OUTPUT
	Done			: BOOL;		(* DataValid Flag is TRUE if Data were available *)
	Err				: BOOL;		(* Err Flag is TRUE if an Error has accured, see Errno for more Details *)
	ErrNo			: UDINT;		(* Contains detailed Error Information *)

	TargetVelocity	: DINT;		(* Target Value *)

END_VAR
VAR
	iStep			: INT;
	ReadObj			: ADSREAD;
	Multiplexor		: UDINT;		(* Gives Index and Subindex of actual Object *)
END_VAR

CASE iStep OF

1:	(* Init *)
	Read := FALSE;
	Done:= FALSE;
	Err := FALSE;
	ErrNo := 0;
	ReadObj(READ := FALSE);
	iStep := 100;

100:	(* Read Object *)
	ReadObj(
		NETID := ADSNetId,
		PORT := 16#1000 + NodeId,
		IDXGRP := 16#60FF,
		IDXOFFS := 0,
		LEN := 4,
		DESTADDR := ADR(TargetVelocity),
		READ := TRUE,
		TMOUT := t#100ms);
	iStep := 101;
101:  ReadObj();
	IF NOT ReadObj.Busy THEN
		iStep := 102 ;
	END_IF
102:	IF ReadObj.Err THEN
		iStep := 0;
		ErrNo := ReadObj.ErrId;
		Multiplexor := 16#60FF00;
		Err := TRUE;
	ELSE
		iStep := 0;
	END_IF;
	Done := TRUE;

ELSE
	IF Read THEN
		iStep := 1;
		Done := FALSE;
	END_IF;
END_CASE;

END_FUNCTION_BLOCK

// POUs/MotionInfo/FB_GetVelocityIs
FUNCTION_BLOCK FB_GetVelocityIs
(*************************************************************************************************************************************
**	maxon motor ag
**	elektronik & systemtechnik
**	all rights reserved
**************************************************************************************************************************************
**	Summary :		Read Actual Value of Velocity
**
**	Remarks : 	
**
**	Created under :	TwinCAT V 2.9.0 (Build 514)
**************************************************************************************************************************************
**	History : 
**	13.10.2003 	| 	san		Beta Version 0.10
**
*************************************************************************************************************************************)
VAR_INPUT
	ADSNetId		: STRING; 	(* Adresses the FC5101 or other Beckhoff CANOpen Masters.
								Can be empty if only local single channel card is present  *)
	NodeId			: INT;		(* Represents the node adress witch is found on Dip Switch of Device *)
	Read			: BOOL;		(* a rising edge start the reading *)

END_VAR
VAR_OUTPUT
	Done			: BOOL;		(* DataValid Flag is TRUE if Data were available *)
	Err				: BOOL;		(* Err Flag is TRUE if an Error has accured, see Errno for more Details *)
	ErrNo			: UDINT;		(* Contains detailed Error Information *)

	VelocityIs		: DINT;		(* Actual Value *)
END_VAR
VAR
	iStep			: INT;
	ReadObj			: ADSREAD;
	Multiplexor		: UDINT;		(* Gives Index and Subindex of actual Object *)
END_VAR

CASE iStep OF

1:	(* Init *)
	Read := FALSE;
	Done := FALSE;
	Err := FALSE;
	ErrNo := 0;
	ReadObj(READ := FALSE);
	iStep := 100;

100:	(* Read Object *)
	ReadObj(
		NETID := ADSNetId,
		PORT := 16#1000 + NodeId,
		IDXGRP := 16#606C,
		IDXOFFS := 0,
		LEN := 4,
		DESTADDR := ADR(VelocityIs),
		READ := TRUE,
		TMOUT := t#100ms);
	iStep := 101;
101:  ReadObj();
	IF NOT ReadObj.Busy THEN
		iStep := 102 ;
	END_IF
102:	IF ReadObj.Err THEN
		iStep := 0;
		ErrNo := ReadObj.ErrId;
		Multiplexor := 16#606C00;
		Err := TRUE;
	ELSE
		iStep := 0;
	END_IF;
	Done := TRUE;

ELSE
	IF Read THEN
		iStep := 1;
		Done := FALSE;
	END_IF;
END_CASE;

END_FUNCTION_BLOCK

// POUs/VelocityMode/FB_GetVelocityMust
FUNCTION_BLOCK FB_GetVelocityMust
(*************************************************************************************************************************************
**	maxon motor ag
**	elektronik & systemtechnik
**	all rights reserved
**************************************************************************************************************************************
**	Summary :		Read Demand Value of Velocity
**
**	Remarks : 	
**
**	Created under :	TwinCAT V 2.9.0 (Build 514)
**************************************************************************************************************************************
**	History : 
**	13.10.2003 	| 	san		Beta Version 0.10
**
*************************************************************************************************************************************)
VAR_INPUT
	ADSNetId		: STRING; 	(* Adresses the FC5101 or other Beckhoff CANOpen Masters.
								Can be empty if only local single channel card is present  *)
	NodeId			: INT;		(* Represents the node adress witch is found on Dip Switch of Device *)
	Read			: BOOL;		(* a rising edge start the reading *)

END_VAR
VAR_OUTPUT
	Done			: BOOL;		(* DataValid Flag is TRUE if Data were available *)
	Err				: BOOL;		(* Err Flag is TRUE if an Error has accured, see Errno for more Details *)
	ErrNo			: UDINT;		(* Contains detailed Error Information *)

	VelocityMust		: DINT;		(* Demand Value *)
END_VAR
VAR
	iStep			: INT;
	ReadObj			: ADSREAD;
	Multiplexor		: UDINT;		(* Gives Index and Subindex of actual Object *)
END_VAR

CASE iStep OF

1:	(* Init *)
	Read := FALSE;
	Done := FALSE;
	Err := FALSE;
	ErrNo := 0;
	ReadObj(READ := FALSE);
	iStep := 100;

100:	(* Read Object *)
	ReadObj(
		NETID := ADSNetId,
		PORT := 16#1000 + NodeId,
		IDXGRP := 16#206B,
		IDXOFFS := 0,
		LEN := 4,
		DESTADDR := ADR(VelocityMust),
		READ := TRUE,
		TMOUT := t#100ms);
	iStep := 101;
101:  ReadObj();
	IF NOT ReadObj.Busy THEN
		iStep := 102 ;
	END_IF
102:	IF ReadObj.Err THEN
		iStep := 0;
		ErrNo := ReadObj.ErrId;
		Multiplexor := 16#206B00;
		Err := TRUE;
	ELSE
		iStep := 0;
	END_IF;
	Done := TRUE;

ELSE
	IF Read THEN
		iStep := 1;
		Done := FALSE;
	END_IF;
END_CASE;

END_FUNCTION_BLOCK

// POUs/ProfileVelocityMode/FB_GetVelocityProfile
FUNCTION_BLOCK FB_GetVelocityProfile
(*************************************************************************************************************************************
**	maxon motor ag
**	elektronik & systemtechnik
**	all rights reserved
**************************************************************************************************************************************
**	Summary :		Get Velocity Profile
**
**	Remarks : 		
**
**	Created under:	TwinCAT V 2.9.0 (Build 514)
**************************************************************************************************************************************
**	History : 
**	13.10.2003 	| 	san		Beta Version 0.10
**
*************************************************************************************************************************************)
VAR_INPUT
	ADSNetId		: STRING; 	(* Adresses the FC5101 or other Beckhoff CANOpen Masters.
								Can be empty if only local single channel card is present  *)
	NodeId			: INT;		(* Represents the node adress witch is found on Dip Switch of Device *)
	Read			: BOOL;		(* a rising edge starts reading *)

END_VAR
VAR_OUTPUT
	Done			: BOOL;		(* Done Flag is set when Function has done *)
	Err				: BOOL;		(* Err Flag is TRUE if an Error has accured, see Errno for more Details *)
	ErrNo			: UDINT;		(* Contains detailed Error Information *)

	ProfileAcceleration: UDINT;		(* Profile Acceleration *)
	ProfileDeceleration: UDINT;		(* Profile Deceleration *)
END_VAR
VAR
	iStep			: INT;
	ReadAcc		: ADSREAD;
	ReadDec		: ADSREAD;
	Multiplexor		: UDINT;		(* Gives Index and Subindex of actual Object *)
END_VAR

CASE iStep OF

1:	(* Init *)
	Read := FALSE;
	Done := FALSE;
	Err := FALSE;
	ErrNo := 0;
	ReadAcc(READ := FALSE);
	ReadDec(READ := FALSE);
	iStep := 100;

100:	(* Profile Acceleration *)
	ReadAcc(
		NETID := ADSNetId,
		PORT := 16#1000 + NodeId,
		IDXGRP := 16#6083,
		IDXOFFS := 0,
		LEN := 4,
		DESTADDR := ADR(ProfileAcceleration),
		READ := TRUE,
		TMOUT := t#100ms);
	iStep := 101;
101:  ReadAcc();
	IF NOT ReadAcc.Busy THEN
		iStep := 102 ;
	END_IF
102:	IF ReadAcc.Err THEN
		iStep := 0;
		ErrNo := ReadAcc.ErrId;
		Multiplexor := 16#608300;
		Err := TRUE;
	ELSE
		iStep := 200;
	END_IF

200:	(* Profile Deceleration *)
	ReadDec(
		NETID := ADSNetId,
		PORT := 16#1000 + NodeId,
		IDXGRP := 16#6084,
		IDXOFFS := 0,
		LEN := 4,
		DESTADDR := ADR(ProfileDeceleration),
		READ := TRUE,
		TMOUT := t#100ms);
	iStep := 201;
201:  ReadDec();
	IF NOT ReadDec.Busy THEN
		iStep := 202 ;
	END_IF
202:	IF ReadDec.Err THEN
		iStep := 0;
		ErrNo := ReadDec.ErrId;
		Multiplexor := 16#608400;
		Err := TRUE;
	ELSE
		iStep := 0;
	END_IF;
	Done := TRUE;

ELSE
	IF Read THEN
		iStep := 1;
		Done := FALSE;
	END_IF;
END_CASE;

END_FUNCTION_BLOCK

// POUs/Configuration/FB_GetVelocityRegulatorGain
FUNCTION_BLOCK FB_GetVelocityRegulatorGain
(*************************************************************************************************************************************
**	maxon motor ag
**	elektronik & systemtechnik
**	all rights reserved
**************************************************************************************************************************************
**	Summary :		Read Velocity Regulator Gains (PI)
**
**	Remarks : 		
**
**	Created under :	TwinCAT V 2.9.0 (Build 514)
**************************************************************************************************************************************
**	History : 
**	13.10.2003 	| 	san		Beta Version 0.10
**
*************************************************************************************************************************************)
VAR_INPUT
	ADSNetId		: STRING; 	(* Adresses the FC5101 or other Beckhoff CANOpen Masters.
								Can be empty if only local single channel card is present  *)
	NodeId			: INT;		(* Represents the node adress witch is found on Dip Switch of Device *)

	Read			: BOOL;		(* a rising edge starts reading *)
END_VAR
VAR_OUTPUT
	Done			: BOOL;		(* Done Flag is set when Function has done *)
	Err				: BOOL;		(* Err Flag is TRUE if an Error has accured, see Errno for more Details *)
	ErrNo			: UDINT;		(* Contains detailed Error Information *)

	P				: UINT;		(* Regulator P - Gain *)
	I				: UINT;		(* Regulator I - Gain  *)
END_VAR
VAR
	iStep			: INT;
	ReadP			: ADSREAD;
	ReadI			: ADSREAD;
	Multiplexor		: UDINT;		(* Gives Index and Subindex of actual Object *)
END_VAR

CASE iStep OF

1:	(* Init *)
	Read := FALSE;
	Done := FALSE;
	Err := FALSE;
	ErrNo := 0;
	ReadP(READ := FALSE);
	ReadI(READ := FALSE);
	iStep := 100;

100:	(* Read P - Gain *)
	ReadP(
		NETID := ADSNetId,
		PORT := 16#1000 + NodeId,
		IDXGRP := 16#60F9,
		IDXOFFS := 1,
		LEN := 2,
		DESTADDR := ADR(P),
		READ := TRUE,
		TMOUT := t#100ms);
	iStep := 101;
101:  ReadP();
	IF NOT ReadP.Busy THEN
		iStep := 102 ;
	END_IF
102:	IF ReadP.Err THEN
		iStep := 0;
		ErrNo := ReadP.ErrId;
		Multiplexor := 16#60F601;
		Err := TRUE;
	ELSE
		iStep := 200;
	END_IF

200:	(* Read I - Gain *)
	ReadI(
		NETID := ADSNetId,
		PORT := 16#1000 + NodeId,
		IDXGRP := 16#60F9,
		IDXOFFS := 2,
		LEN := 2,
		DESTADDR := ADR(I),
		READ := TRUE,
		TMOUT := t#100ms);
	iStep := 201;
201:  ReadI();
	IF NOT ReadI.Busy THEN
		iStep := 202 ;
	END_IF
202:	IF ReadI.Err THEN
		iStep := 0;
		ErrNo := ReadI.ErrId;
		Multiplexor := 16#60F602;
		Err := TRUE;
	ELSE
		iStep := 0;
	END_IF;
	Done := TRUE;

ELSE
	IF Read THEN
		iStep := 1;
	END_IF;
END_CASE;

END_FUNCTION_BLOCK

// POUs/Utilities/FB_GetVersion
FUNCTION_BLOCK FB_GetVersion
(*************************************************************************************************************************************
**	maxon motor ag
**	elektronik & systemtechnik
**	all rights reserved
**************************************************************************************************************************************
**	Summary :		Reads the Hardware-, Software- , Application Version and Application Number
**
**	Remarks : 	
**
**	Created under :	TwinCAT V 2.9.0 (Build 514)
**************************************************************************************************************************************
**	History : 
**	13.10.2003 	| 	san		Beta Version 0.10
**
*************************************************************************************************************************************)
VAR_INPUT
	ADSNetId		: STRING; 	(* Adresses the FC5101 or other Beckhoff CANOpen Masters.
								Can be empty if only local single channel card is present  *)
	NodeId			: INT;		(* Represents the node adress witch is found on Dip Switch of Device *)
	Read			: BOOL;		(* a rising edge start the reading *)
END_VAR
VAR_OUTPUT
	Done			: BOOL;		(* DataValid Flag is TRUE if Data were available *)
	Err				: BOOL;		(* Err Flag is TRUE if an Error has accured, see Errno for more Details *)
	ErrNo			: UDINT;		(* Contains detailed Error Information *)

	HardwareVersion	: UINT;		(* Hardware Version *)
	SoftwareVersion	: UINT;		(* Software Version *)
	ApplicationVersion: UINT;		(* Application Version *)
	ApplicationNumber: UINT;		(* Application Number *)
END_VAR
VAR
	iStep			: INT;
	ReadHw			: ADSREAD;
	ReadSw			: ADSREAD;
	ReadApp		: ADSREAD;
	ReadAppNo		: ADSREAD;
	Multiplexor		: UDINT;		(* Gives Index and Subindex of actual Object *)
END_VAR

CASE iStep OF

1:	(* Init *)
	Read := FALSE;
	Done := FALSE;
	Err := FALSE;
	ErrNo := 0;
	ReadHw(READ := FALSE);
	ReadSw(READ := FALSE);
	ReadApp(READ := FALSE);
	ReadAppNo(READ := FALSE);
	iStep := 100;

100:	(* Read Hardware Version *)
	ReadHw(
		NETID := ADSNetId,
		PORT := 16#1000 + NodeId,
		IDXGRP := 16#2003,
		IDXOFFS := 2,
		LEN := 2,
		DESTADDR := ADR(HardwareVersion),
		READ := TRUE,
		TMOUT := t#100ms);
	iStep := 101;
101:  ReadHw();
	IF NOT ReadHw.Busy THEN
		iStep := 102 ;
	END_IF
102:	IF ReadHw.Err THEN
		iStep := 0;
		ErrNo := ReadHw.ErrId;
		Multiplexor := 16#200302;
		Err := TRUE;
	ELSE
		iStep := 200;
	END_IF

200:	(* Read Software Version *)
	ReadSw(
		NETID := ADSNetId,
		PORT := 16#1000 + NodeId,
		IDXGRP := 16#2003,
		IDXOFFS := 1,
		LEN := 2,
		DESTADDR := ADR(SoftwareVersion),
		READ := TRUE,
		TMOUT := t#100ms);
	iStep := 201;
201:  ReadSw();
	IF NOT ReadSw.Busy THEN
		iStep := 202 ;
	END_IF
202:	IF ReadSw.Err THEN
		iStep := 0;
		ErrNo := ReadSw.ErrId;
		Multiplexor := 16#200301;
		Err := TRUE;
	ELSE
		iStep := 300;
	END_IF
300:	(* Read Application Version *)
	ReadApp(
		NETID := ADSNetId,
		PORT := 16#1000 + NodeId,
		IDXGRP := 16#2003,
		IDXOFFS := 4,
		LEN := 2,
		DESTADDR := ADR(ApplicationVersion),
		READ := TRUE,
		TMOUT := t#100ms);
	iStep := 301;
301:  ReadApp();
	IF NOT ReadApp.Busy THEN
		iStep := 302 ;
	END_IF
302:	IF ReadApp.Err THEN
		iStep := 0;
		ErrNo := ReadApp.ErrId;
		Multiplexor := 16#200304;
		Err := TRUE;
	ELSE
		iStep := 400;
	END_IF
400:	(* Read Application Number *)
	ReadAppNo(
		NETID := ADSNetId,
		PORT := 16#1000 + NodeId,
		IDXGRP := 16#2003,
		IDXOFFS := 3,
		LEN := 2,
		DESTADDR := ADR(ApplicationNumber),
		READ := TRUE,
		TMOUT := t#100ms);
	iStep := 401;
401:  ReadAppNo();
	IF NOT ReadAppNo.Busy THEN
		iStep := 402 ;
	END_IF
402:	IF ReadAppNo.Err THEN
		iStep := 0;
		ErrNo := ReadAppNo.ErrId;
		Multiplexor := 16#200303;
		Err := TRUE;
	ELSE
		iStep := 0;
	END_IF;
	Done := TRUE;

ELSE
	IF Read THEN
		iStep := 1;
		Done := FALSE;
	END_IF;
END_CASE;

END_FUNCTION_BLOCK

// POUs/ProfilePositionMode/FB_HaltPositionMovement
FUNCTION_BLOCK FB_HaltPositionMovement
(*************************************************************************************************************************************
**	maxon motor ag
**	elektronik & systemtechnik
**	all rights reserved
**************************************************************************************************************************************
**	Summary :		Halt with Position Profile set by SetPositionProfile
**
**	Remarks : 		
**
**	Created under:	TwinCAT V 2.9.0 (Build 514)
**************************************************************************************************************************************
**	History : 
**	13.10.2003 	| 	san		Beta Version 0.10
**
*************************************************************************************************************************************)
VAR_INPUT
	ADSNetId		: STRING; 	(* Adresses the FC5101 or other Beckhoff CANOpen Masters.
								Can be empty if only local single channel card is present  *)
	NodeId			: INT;		(*Represents the node adress witch is found on Dip Switch of Device *)

	Write			: BOOL;		(* a rising edge starts writing *)
END_VAR
VAR_OUTPUT
	Done			: BOOL;		(* Done Flag is set when Function has done *)
	Err				: BOOL;		(* Err Flag is TRUE if an Error has accured, see Errno for more Details *)
	ErrNo			: UDINT;		(* Contains detailed Error Information *)
END_VAR
VAR
	iStep			: INT;
	WriteCw			: ADSWRITE;
	uiControlword		: UINT;
	Multiplexor		: UDINT;		(* Gives Index and Subindex of actual Object *)
END_VAR

CASE iStep OF

1:	(* Init *)
	Write := FALSE;
	Done := FALSE;
	Err := FALSE;
	ErrNo := 0;
	WriteCw(WRITE := FALSE);
	iStep := 100;

100:	(* Controlword *)
	uiControlword := 16#010F;
	WriteCw(
		NETID := ADSNetId,
		PORT := 16#1000 + NodeId,
		IDXGRP := 16#6040,
		IDXOFFS := 0,
		LEN := 2,
		SRCADDR := ADR(uiControlword),
		WRITE := TRUE,
		TMOUT := t#100ms);
	iStep := 101;
101:  WriteCw();
	IF NOT WriteCw.Busy THEN
		iStep := 102 ;
	END_IF
102:	IF WriteCw.Err THEN
		iStep := 0;
		ErrNo := WriteCw.ErrId;
		Multiplexor := 16#604000;
		Err := TRUE;
	ELSE
		iStep := 0;
	END_IF;
	Done := TRUE;

ELSE
	IF Write THEN
		iStep := 1;
		Done := FALSE;
	END_IF;
END_CASE;

END_FUNCTION_BLOCK

// POUs/ProfileVelocityMode/FB_HaltVelocityMovement
FUNCTION_BLOCK FB_HaltVelocityMovement
(*************************************************************************************************************************************
**	maxon motor ag
**	elektronik & systemtechnik
**	all rights reserved
**************************************************************************************************************************************
**	Summary :		Halt with Position Profile set by SetPositionProfile
**
**	Remarks : 		
**
**	Created under:	TwinCAT V 2.9.0 (Build 514)
**************************************************************************************************************************************
**	History : 
**	13.10.2003 	| 	san		Beta Version 0.10
**
*************************************************************************************************************************************)
VAR_INPUT
	ADSNetId		: STRING; 	(* Adresses the FC5101 or other Beckhoff CANOpen Masters.
								Can be empty if only local single channel card is present  *)
	NodeId			: INT;		(*Represents the node adress witch is found on Dip Switch of Device *)

	Write			: BOOL;		(* a rising edge starts writing *)
END_VAR
VAR_OUTPUT
	Done			: BOOL;		(* Done Flag is set when Function has done *)
	Err				: BOOL;		(* Err Flag is TRUE if an Error has accured, see Errno for more Details *)
	ErrNo			: UDINT;		(* Contains detailed Error Information *)
END_VAR
VAR
	iStep			: INT;
	WriteCw			: ADSWRITE;
	uiControlword		: UINT;
	Multiplexor		: UDINT;		(* Gives Index and Subindex of actual Object *)
END_VAR

CASE iStep OF

1:	(* Init *)
	Write := FALSE;
	Done := FALSE;
	Err := FALSE;
	ErrNo := 0;
	WriteCw(WRITE := FALSE);
	iStep := 100;

100:	(* Controlword *)
	uiControlword := 16#010F;
	WriteCw(
		NETID := ADSNetId,
		PORT := 16#1000 + NodeId,
		IDXGRP := 16#6040,
		IDXOFFS := 0,
		LEN := 2,
		SRCADDR := ADR(uiControlword),
		WRITE := TRUE,
		TMOUT := t#100ms);
	iStep := 101;
101:  WriteCw();
	IF NOT WriteCw.Busy THEN
		iStep := 102 ;
	END_IF
102:	IF WriteCw.Err THEN
		iStep := 0;
		ErrNo := WriteCw.ErrId;
		Multiplexor := 16#604000;
		Err := TRUE;
	ELSE
		iStep := 0;
	END_IF;
	Done := TRUE;

ELSE
	IF Write THEN
		iStep := 1;
		Done := FALSE;
	END_IF;
END_CASE;

END_FUNCTION_BLOCK

// POUs/ProfilePositionMode/FB_MoveToPosition
FUNCTION_BLOCK FB_MoveToPosition
(*************************************************************************************************************************************
**	maxon motor ag
**	elektronik & systemtechnik
**	all rights reserved
**************************************************************************************************************************************
**	Summary :		Move Point to Point 
**
**	Remarks : 		
**
**	Created under:	TwinCAT V 2.9.0 (Build 514)
**************************************************************************************************************************************
**	History : 
**	13.10.2003 	| 	san		Beta Version 0.10
**
*************************************************************************************************************************************)
VAR_INPUT
	ADSNetId		: STRING; 	(* Adresses the FC5101 or other Beckhoff CANOpen Masters.
								Can be empty if only local single channel card is present  *)
	NodeId			: INT;		(*Represents the node adress witch is found on Dip Switch of Device *)

	Write			: BOOL;		(* a rising edge starts writing *)

	TargetPosition	: DINT;		(* Target Position *)
	Absolut			: BOOL;		(* 	TRUE :	Starts a Point to Point Movement to Absolute Position  (relative to Home)
									FALSE:	Starts a Point to Point Movement to Relative Position (relative to Actual Position)*)

END_VAR
VAR_OUTPUT
	Done			: BOOL;		(* Done Flag is set when Function has done *)
	Err				: BOOL;		(* Err Flag is TRUE if an Error has accured, see Errno for more Details *)
	ErrNo			: UDINT;		(* Contains detailed Error Information *)
END_VAR
VAR
	iStep			: INT;
	WritePos			: ADSWRITE;
	WriteCw			: ADSWRITE;
	uiControlword		: UINT;
	Multiplexor		: UDINT;		(* Gives Index and Subindex of actual Object *)
END_VAR

CASE iStep OF

1:	(* Init *)
	Write := FALSE;
	Done := FALSE;
	Err := FALSE;
	ErrNo := 0;
	WritePos(WRITE := FALSE);
	WriteCw(WRITE := FALSE);
	iStep := 100;

100:	(* Target Position *)
	WritePos(
		NETID := ADSNetId,
		PORT := 16#1000 + NodeId,
		IDXGRP := 16#607A,
		IDXOFFS := 0,
		LEN := 4,
		SRCADDR := ADR(TargetPosition),
		WRITE := TRUE,
		TMOUT := t#100ms);
	iStep := 101;
101:  WritePos();
	IF NOT WritePos.Busy THEN
		iStep := 102 ;
	END_IF
102:	IF WritePos.Err THEN
		iStep := 0;
		ErrNo := WritePos.ErrId;
		Multiplexor := 16#607A00;
		Err := TRUE;
	ELSE
		iStep := 200;
	END_IF

200:	(* Controlword *)
	IF Absolut THEN
		uiControlword := 16#001F;
	ELSE
		uiControlword := 16#005F;
	END_IF;
	WriteCw(
		NETID := ADSNetId,
		PORT := 16#1000 + NodeId,
		IDXGRP := 16#6040,
		IDXOFFS := 0,
		LEN := 2,
		SRCADDR := ADR(uiControlword),
		WRITE := TRUE,
		TMOUT := t#100ms);
	iStep := 201;
201:  WriteCw ();
	IF NOT WriteCw.Busy THEN
		iStep := 202 ;
	END_IF
202:	IF WriteCw.Err THEN
		iStep := 0;
		ErrNo := WriteCw.ErrId;
		Multiplexor := 16#604000;
		Err := TRUE;
	ELSE
		iStep := 0;
	END_IF;
	Done := TRUE;

ELSE
	IF Write THEN
		iStep := 1;
		Done := FALSE ;
	END_IF;
END_CASE;

END_FUNCTION_BLOCK

// POUs/ProfileVelocityMode/FB_MoveWithVelocity
FUNCTION_BLOCK FB_MoveWithVelocity
(*************************************************************************************************************************************
**	maxon motor ag
**	elektronik & systemtechnik
**	all rights reserved
**************************************************************************************************************************************
**	Summary :		Move with Target Velocity
**
**	Remarks : 		
**
**	Created under:	TwinCAT V 2.9.0 (Build 514)
**************************************************************************************************************************************
**	History : 
**	13.10.2003 	| 	san		Beta Version 0.10
**
*************************************************************************************************************************************)
VAR_INPUT
	ADSNetId		: STRING; 	(* Adresses the FC5101 or other Beckhoff CANOpen Masters.
								Can be empty if only local single channel card is present  *)
	NodeId			: INT;		(* Represents the node adress witch is found on Dip Switch of Device *)
	Write			: BOOL;		(* a rising edge starts writing *)

	TargetVelocity	: DINT;		(* Target Velocity *)
END_VAR
VAR_OUTPUT
	Done			: BOOL;		(* Done Flag is set when Function has done *)
	Err				: BOOL;		(* Err Flag is TRUE if an Error has accured, see Errno for more Details *)
	ErrNo			: UDINT;		(* Contains detailed Error Information *)
END_VAR
VAR
	iStep			: INT;
	WriteVel			: ADSWRITE;
	WriteCw			: ADSWRITE;
	uiControlword		: UINT			:= 16#000F;
	Multiplexor		: UDINT;		(* Gives Index and Subindex of actual Object *)
END_VAR

CASE iStep OF

1:	(* Init *)
	Write := FALSE;
	Done := FALSE;
	Err := FALSE;
	ErrNo := 0;
	WriteVel(WRITE := FALSE);
	WriteCw(WRITE := FALSE);
	iStep := 100;

100:	(* Target Velocity *)
	WriteVel(
		NETID := ADSNetId,
		PORT := 16#1000 + NodeId,
		IDXGRP := 16#60FF,
		IDXOFFS := 0,
		LEN := 4,
		SRCADDR := ADR(TargetVelocity),
		WRITE := TRUE,
		TMOUT := t#100ms);
	iStep := 101;
101:  WriteVel();
	IF NOT WriteVel.Busy THEN
		iStep := 102 ;
	END_IF
102:	IF WriteVel.Err THEN
		iStep := 0;
		ErrNo := WriteVel.ErrId;
		Multiplexor := 16#60FF00;
		Err := TRUE;
	ELSE
		iStep := 200;
	END_IF

200:	(* Controlword *)
	WriteCw(
		NETID := ADSNetId,
		PORT := 16#1000 + NodeId,
		IDXGRP := 16#6040,
		IDXOFFS := 0,
		LEN := 2,
		SRCADDR := ADR(uiControlword),
		WRITE := TRUE,
		TMOUT := t#100ms);
	iStep := 201;
201:  WriteCw();
	IF NOT WriteCw.Busy THEN
		iStep := 202 ;
	END_IF
202:	IF WriteCw.Err THEN
		iStep := 0;
		ErrNo := WriteCw.ErrId;
		Multiplexor := 16#604000;
		Err := TRUE;
	ELSE
		iStep := 0;
	END_IF;
	Done := TRUE;

ELSE
	IF Write THEN
		iStep := 1;
		Done := FALSE;
	END_IF;
END_CASE;

END_FUNCTION_BLOCK

// POUs/Utilities/FB_Restore
FUNCTION_BLOCK FB_Restore
(*************************************************************************************************************************************
**	maxon motor ag
**	elektronik & systemtechnik
**	all rights reserved
**************************************************************************************************************************************
**	Summary :		Restore all system parameters
**
**	Remarks : 	
**
**	Created under :	TwinCAT V 2.9.0 (Build 514)
**************************************************************************************************************************************
**	History : 
**	13.10.2003 	| 	san		Beta Version 0.10
**
*************************************************************************************************************************************)
VAR_INPUT
	ADSNetId		: STRING; 	(* Adresses the FC5101 or other Beckhoff CANOpen Masters.
								Can be empty if only local single channel card is present  *)
	NodeId			: INT;		(* Represents the node adress witch is found on Dip Switch of Device *)
	Write			: BOOL;		(* a rising edge starts writing *)

END_VAR
VAR_OUTPUT
	Done			: BOOL;		(* Done Flag is set when Function has done *)
	Err				: BOOL;		(* Err Flag is TRUE if an Error has accured, see Errno for more Details *)
	ErrNo			: UDINT;		(* Contains detailed Error Information *)
END_VAR
VAR
	iStep			: INT;
	WriteObj			: ADSWRITE;
	udiData: 			UDINT			:= 16#64616F6C;
	ODIdx: 			BOOL;
	Multiplexor		: UDINT;		(* Gives Index and Subindex of actual Object *)
END_VAR

CASE iStep OF

1:	(* Init *)
	Write := FALSE;
	Done := FALSE;
	Err := FALSE;
	ErrNo := 0;
	WriteObj(WRITE := FALSE);
	iStep := 100;

100:	(* Read Object *)
	WriteObj(
		NETID := ADSNetId,
		PORT := 16#1000 + NodeId,
		IDXGRP := 16#1011,
		IDXOFFS := 1,
		LEN := 4,
		SRCADDR := ADR(udiData),
		WRITE := TRUE,
		TMOUT := t#100ms);
	iStep := 101;
101:  WriteObj();
	IF NOT WriteObj.Busy THEN
		iStep := 102 ;
	END_IF
102:	IF WriteObj.Err THEN
		iStep := 0;
		ErrNo := WriteObj.ErrId;
		Multiplexor := 16#101001;
		Err := TRUE;
	ELSE
		iStep := 0;
	END_IF;
	Done := TRUE;

ELSE
	IF Write THEN
		iStep := 1;
		Done := FALSE;
	END_IF;
END_CASE;

END_FUNCTION_BLOCK

// POUs/InputsOutputs/FB_SetAllDigitalOutputs
FUNCTION_BLOCK FB_SetAllDigitalOutputs
(*************************************************************************************************************************************
**	maxon motor ag
**	elektronik & systemtechnik
**	all rights reserved
**************************************************************************************************************************************
**	Summary :		Set all Digital Outputs
**
**	Remarks : 	
**
**	Created under :	TwinCAT V 2.9.0 (Build 514)
**************************************************************************************************************************************
**	History : 
**	16.09.2003 	| 	san		Beta Version 0.10
**	21.11.2003	|	san		Beta Version 0.20 firmware changes
**
*************************************************************************************************************************************)
VAR_INPUT
	ADSNetId		: STRING; 	(* Adresses the FC5101 or other Beckhoff CANOpen Masters.
								Can be empty if only local single channel card is present  *)
	NodeId			: INT;		(* Represents the node adress witch is found on Dip Switch of Device *)
	Write			: BOOL;		(* a rising edge starts writing *)

	Outputs			: UINT;		(* Outputs to set *)


END_VAR
VAR_OUTPUT
	Done			: BOOL;		(* Done Flag is set when Function has done *)
	Err				: BOOL;		(* Err Flag is TRUE if an Error has accured, see Errno for more Details *)
	ErrNo			: UDINT;		(* Contains detailed Error Information *)
END_VAR
VAR
	iStep			: INT;
	WriteObj			: ADSWRITE;
	ODIdx			: UINT			:= 16#2078;
	ODSubidx		: UINT			:= 1;
	Multiplexor		: UDINT;		(* Gives Index and Subindex of actual Object *)
END_VAR

CASE iStep OF

1:	(* Init *)
	Write := FALSE;
	Done := FALSE;
	Err := FALSE;
	ErrNo := 0;
	WriteObj(WRITE := FALSE);
	iStep := 100;

100:	(* Write Object *)
	WriteObj(
		NETID := ADSNetId,
		PORT := 16#1000 + NodeId,
		IDXGRP := ODIdx,
		IDXOFFS := ODSubidx,
		LEN := 2,
		SRCADDR := ADR(Outputs),
		WRITE := TRUE,
		TMOUT := t#100ms);
	iStep := 101;
101:  WriteObj();
	IF NOT WriteObj.Busy THEN
		iStep := 102 ;
	END_IF
102:	IF WriteObj.Err THEN
		iStep := 0;
		ErrNo := WriteObj.ErrId;
		Multiplexor := ODIdx * 256; (* Shift of 8 *)
		Multiplexor := Multiplexor + ODSubidx;
		Err := TRUE;
	ELSE
		iStep := 0;
	END_IF;
	Done := TRUE;

ELSE
	IF Write THEN
		iStep := 1;
		Done := FALSE;
	END_IF;
END_CASE;

END_FUNCTION_BLOCK

